gfCNCPoint2[2423] = {X 419.9424, Y 96.5448, Z -2.1667, A 0.000, B 0.000, C 0.000 }
gfCNCPoint2[2424] = {X 419.9467, Y 97.0649, Z -2.1667, A 0.000, B 0.000, C 0.000 }
gfCNCPoint2[2425] = {X 419.9467, Y 98.0000, Z -2.1667, A 0.000, B 0.000, C 0.000 }
gfCNCPoint2[2426] = {X 419.8404, Y 98.9435, Z -2.1667, A 0.000, B 0.000, C 0.000 }
gfCNCPoint2[2427] = {X 419.5268, Y 99.8397, Z -2.1667, A 0.000, B 0.000, C 0.000 }
gfCNCPoint2[2428] = {X 419.0217, Y 100.6436, Z -2.1667, A 0.000, B 0.000, C 0.000 }
gfCNCPoint2[2429] = {X 418.3503, Y 101.3150, Z -2.1667, A 0.000, B 0.000, C 0.000 }
gfCNCPoint2[2430] = {X 417.5464, Y 101.8201, Z -2.1667, A 0.000, B 0.000, C 0.000 }
gfCNCPoint2[2431] = {X 416.6502, Y 102.1337, Z -2.1667, A 0.000, B 0.000, C 0.000 }
gfCNCPoint2[2432] = {X 415.7067, Y 102.2400, Z -2.1667, A 0.000, B 0.000, C 0.000 }
gfCNCPoint2[2433] = {X 396.4059, Y 102.2400, Z -2.1667, A 0.000, B 0.000, C 0.000 }
gfCNCPoint2[2434] = {X 395.4625, Y 102.1337, Z -2.1667, A 0.000, B 0.000, C 0.000 }
gfCNCPoint2[2435] = {X 394.5663, Y 101.8201, Z -2.1667, A 0.000, B 0.000, C 0.000 }
gfCNCPoint2[2436] = {X 393.7624, Y 101.3150, Z -2.1667, A 0.000, B 0.000, C 0.000 }
gfCNCPoint2[2437] = {X 393.0910, Y 100.6436, Z -2.1667, A 0.000, B 0.000, C 0.000 }
gfCNCPoint2[2438] = {X 392.5858, Y 99.8397, Z -2.1667, A 0.000, B 0.000, C 0.000 }
gfCNCPoint2[2439] = {X 392.2723, Y 98.9435, Z -2.1667, A 0.000, B 0.000, C 0.000 }
gfCNCPoint2[2440] = {X 392.1659, Y 98.0000, Z -2.1667, A 0.000, B 0.000, C 0.000 }
gfCNCPoint2[2441] = {X 392.1659, Y 97.0659, Z -2.1667, A 0.000, B 0.000, C 0.000 }
gfCNCPoint2[2442] = {X 392.2718, Y 96.1245, Z -2.1667, A 0.000, B 0.000, C 0.000 }
gfCNCPoint2[2443] = {X 392.5840, Y 95.2301, Z -2.1667, A 0.000, B 0.000, C 0.000 }
gfCNCPoint2[2444] = {X 393.0870, Y 94.4274, Z -2.1667, A 0.000, B 0.000, C 0.000 }
gfCNCPoint2[2445] = {X 393.7556, Y 93.7563, Z -2.1667, A 0.000, B 0.000, C 0.000 }
gfCNCPoint2[2446] = {X 394.5566, Y 93.2505, Z -2.1667, A 0.000, B 0.000, C 0.000 }
gfCNCPoint2[2447] = {X 395.4499, Y 92.9351, Z -2.1667, A 0.000, B 0.000, C 0.000 }
gfCNCPoint2[2448] = {X 396.3909, Y 92.8260, Z -2.1667, A 0.000, B 0.000, C 0.000 }
gfCNCPoint2[2449] = {X 397.3487, Y 92.7854, Z -2.1667, A 0.000, B 0.000, C 0.000 }
gfCNCPoint2[2450] = {X 398.3031, Y 92.6947, Z -2.1667, A 0.000, B 0.000, C 0.000 }
gfCNCPoint2[2451] = {X 398.9716, Y 92.5328, Z -2.1667, A 0.000, B 0.000, C 0.000 }
gfCNCPoint2[2452] = {X 399.5871, Y 92.2258, Z -2.1667, A 0.000, B 0.000, C 0.000 }
gfCNCPoint2[2453] = {X 413.8427, Y 83.0964, Z -2.1667, A 0.000, B 0.000, C 0.000 }
gfCNCPoint2[2454] = {X 411.6855, Y 79.7280, Z -2.1667, A 0.000, B 0.000, C 0.000 }
gfCNCPoint2[2455] = {X 413.8858, Y 83.1638, Z -2.1667, A 0.000, B 0.000, C 0.000 }
gfCNCPoint2[2456] = {X 428.4059, Y 73.8650, Z -2.1667, A 0.000, B 0.000, C 0.000 }
gfCNCPoint2[2457] = {X 403.8140, Y 64.2159, Z -2.1667, A 0.000, B 0.000, C 0.000 }
gfCNCPoint2[2458] = {X 402.1005, Y 63.6486, Z -2.1667, A 0.000, B 0.000, C 0.000 }
gfCNCPoint2[2459] = {X 400.3349, Y 63.2731, Z -2.1667, A 0.000, B 0.000, C 0.000 }
gfCNCPoint2[2460] = {X 398.5388, Y 63.0940, Z -2.1667, A 0.000, B 0.000, C 0.000 }
gfCNCPoint2[2461] = {X 397.6210, Y 62.9872, Z -2.1667, A 0.000, B 0.000, C 0.000 }
gfCNCPoint2[2462] = {X 396.7495, Y 62.6805, Z -2.1667, A 0.000, B 0.000, C 0.000 }
gfCNCPoint2[2463] = {X 395.9671, Y 62.1889, Z -2.1667, A 0.000, B 0.000, C 0.000 }
gfCNCPoint2[2464] = {X 395.3125, Y 61.5368, Z -2.1667, A 0.000, B 0.000, C 0.000 }
gfCNCPoint2[2465] = {X 394.8180, Y 60.7563, Z -2.1667, A 0.000, B 0.000, C 0.000 }
gfCNCPoint2[2466] = {X 394.5081, Y 59.8858, Z -2.1667, A 0.000, B 0.000, C 0.000 }
gfCNCPoint2[2467] = {X 394.3979, Y 58.9684, Z -2.1667, A 0.000, B 0.000, C 0.000 }
gfCNCPoint2[2468] = {X 394.3977, Y 58.0000, Z -2.1667, A 0.000, B 0.000, C 0.000 }
gfCNCPoint2[2469] = {X 394.5020, Y 57.0743, Z -2.1667, A 0.000, B 0.000, C 0.000 }
gfCNCPoint2[2470] = {X 394.8097, Y 56.1950, Z -2.1667, A 0.000, B 0.000, C 0.000 }
gfCNCPoint2[2471] = {X 395.3053, Y 55.4063, Z -2.1667, A 0.000, B 0.000, C 0.000 }
gfCNCPoint2[2472] = {X 395.9640, Y 54.7476, Z -2.1667, A 0.000, B 0.000, C 0.000 }
gfCNCPoint2[2473] = {X 396.7528, Y 54.2520, Z -2.1667, A 0.000, B 0.000, C 0.000 }
gfCNCPoint2[2474] = {X 397.6320, Y 53.9443, Z -2.1667, A 0.000, B 0.000, C 0.000 }
gfCNCPoint2[2475] = {X 398.5577, Y 53.8400, Z -2.1667, A 0.000, B 0.000, C 0.000 }
gfCNCPoint2[2476] = {X 419.4886, Y 53.8400, Z -2.1667, A 0.000, B 0.000, C 0.000 }
gfCNCPoint2[2477] = {X 420.4143, Y 53.9443, Z -2.1667, A 0.000, B 0.000, C 0.000 }
gfCNCPoint2[2478] = {X 421.2936, Y 54.2520, Z -2.1667, A 0.000, B 0.000, C 0.000 }
gfCNCPoint2[2479] = {X 422.0823, Y 54.7476, Z -2.1667, A 0.000, B 0.000, C 0.000 }
gfCNCPoint2[2480] = {X 422.7410, Y 55.4063, Z -2.1667, A 0.000, B 0.000, C 0.000 }
gfCNCPoint2[2481] = {X 423.2366, Y 56.1950, Z -2.1667, A 0.000, B 0.000, C 0.000 }
gfCNCPoint2[2482] = {X 423.5443, Y 57.0743, Z -2.1667, A 0.000, B 0.000, C 0.000 }
gfCNCPoint2[2483] = {X 423.6486, Y 58.0000, Z -2.1667, A 0.000, B 0.000, C 0.000 }
gfCNCPoint2[2484] = {X 423.6486, Y 58.3421, Z -2.1667, A 0.000, B 0.000, C 0.000 }
gfCNCPoint2[2485] = {X 429.5531, Y 60.6433, Z -2.1667, A 0.000, B 0.000, C 0.000 }
gfCNCPoint2[2486] = {X 458.0211, Y 71.9378, Z -2.1667, A 0.000, B 0.000, C 0.000 }
gfCNCPoint2[2487] = {X 458.0212, Y 63.0709, Z -2.1667, A 0.000, B 0.000, C 0.000 }
gfCNCPoint2[2488] = {X 457.9189, Y 63.0588, Z -2.1667, A 0.000, B 0.000, C 0.000 }
gfCNCPoint2[2489] = {X 457.8169, Y 63.0441, Z -2.1667, A 0.000, B 0.000, C 0.000 }
gfCNCPoint2[2490] = {X 456.8792, Y 62.7822, Z -2.1667, A 0.000, B 0.000, C 0.000 }
gfCNCPoint2[2491] = {X 456.0281, Y 62.3095, Z -2.1667, A 0.000, B 0.000, C 0.000 }
gfCNCPoint2[2492] = {X 455.3102, Y 61.6519, Z -2.1667, A 0.000, B 0.000, C 0.000 }
gfCNCPoint2[2493] = {X 454.7647, Y 60.8455, Z -2.1667, A 0.000, B 0.000, C 0.000 }
gfCNCPoint2[2494] = {X 454.4217, Y 59.9343, Z -2.1667, A 0.000, B 0.000, C 0.000 }
gfCNCPoint2[2495] = {X 454.2997, Y 58.9684, Z -2.1667, A 0.000, B 0.000, C 0.000 }
gfCNCPoint2[2496] = {X 454.2996, Y 58.0000, Z -2.1667, A 0.000, B 0.000, C 0.000 }
gfCNCPoint2[2497] = {X 454.4039, Y 57.0743, Z -2.1667, A 0.000, B 0.000, C 0.000 }
gfCNCPoint2[2498] = {X 454.7116, Y 56.1950, Z -2.1667, A 0.000, B 0.000, C 0.000 }
gfCNCPoint2[2499] = {X 455.2072, Y 55.4063, Z -2.1667, A 0.000, B 0.000, C 0.000 }
gfCNCPoint2[2500] = {X 455.8659, Y 54.7476, Z -2.1667, A 0.000, B 0.000, C 0.000 }
gfCNCPoint2[2501] = {X 456.6546, Y 54.2520, Z -2.1667, A 0.000, B 0.000, C 0.000 }
gfCNCPoint2[2502] = {X 457.5339, Y 53.9443, Z -2.1667, A 0.000, B 0.000, C 0.000 }
gfCNCPoint2[2503] = {X 458.4596, Y 53.8400, Z -2.1667, A 0.000, B 0.000, C 0.000 }
gfCNCPoint2[2504] = {X 475.0000, Y 53.8400, Z -2.1667, A 0.000, B 0.000, C 0.000 }
gfCNCPoint2[2505] = {X 475.9257, Y 53.9443, Z -2.1667, A 0.000, B 0.000, C 0.000 }
gfCNCPoint2[2506] = {X 476.8050, Y 54.2520, Z -2.1667, A 0.000, B 0.000, C 0.000 }
gfCNCPoint2[2507] = {X 477.5937, Y 54.7476, Z -2.1667, A 0.000, B 0.000, C 0.000 }
gfCNCPoint2[2508] = {X 478.2524, Y 55.4063, Z -2.1667, A 0.000, B 0.000, C 0.000 }
gfCNCPoint2[2509] = {X 478.7480, Y 56.1950, Z -2.1667, A 0.000, B 0.000, C 0.000 }
gfCNCPoint2[2510] = {X 479.0557, Y 57.0743, Z -2.1667, A 0.000, B 0.000, C 0.000 }
gfCNCPoint2[2511] = {X 479.1600, Y 58.0000, Z -2.1667, A 0.000, B 0.000, C 0.000 }
gfCNCPoint2[2512] = {X 479.1600, Y 58.9342, Z -2.1667, A 0.000, B 0.000, C 0.000 }
gfCNCPoint2[2513] = {X 479.0692, Y 59.7985, Z -2.1667, A 0.000, B 0.000, C 0.000 }
gfCNCPoint2[2514] = {X 478.8008, Y 60.6250, Z -2.1667, A 0.000, B 0.000, C 0.000 }
gfCNCPoint2[2515] = {X 478.3666, Y 61.3777, Z -2.1667, A 0.000, B 0.000, C 0.000 }
gfCNCPoint2[2516] = {X 477.7855, Y 62.0238, Z -2.1667, A 0.000, B 0.000, C 0.000 }
gfCNCPoint2[2517] = {X 477.0828, Y 62.5351, Z -2.1667, A 0.000, B 0.000, C 0.000 }
gfCNCPoint2[2518] = {X 476.2893, Y 62.8892, Z -2.1667, A 0.000, B 0.000, C 0.000 }
gfCNCPoint2[2519] = {X 475.4395, Y 63.0708, Z -2.1667, A 0.000, B 0.000, C 0.000 }
gfCNCPoint2[2520] = {X 475.4399, Y 92.8982, Z -2.1667, A 0.000, B 0.000, C 0.000 }
gfCNCPoint2[2521] = {X 475.8913, Y 93.0052, Z -2.1667, A 0.000, B 0.000, C 0.000 }
gfCNCPoint2[2522] = {X 476.3356, Y 93.1389, Z -2.1667, A 0.000, B 0.000, C 0.000 }
gfCNCPoint2[2523] = {X 477.1173, Y 93.4941, Z -2.1667, A 0.000, B 0.000, C 0.000 }
gfCNCPoint2[2524] = {X 477.8089, Y 94.0030, Z -2.1667, A 0.000, B 0.000, C 0.000 }
gfCNCPoint2[2525] = {X 478.3804, Y 94.6438, Z -2.1667, A 0.000, B 0.000, C 0.000 }
gfCNCPoint2[2526] = {X 478.8072, Y 95.3889, Z -2.1667, A 0.000, B 0.000, C 0.000 }
gfCNCPoint2[2527] = {X 479.0708, Y 96.2060, Z -2.1667, A 0.000, B 0.000, C 0.000 }
gfCNCPoint2[2528] = {X 479.1600, Y 97.0600, Z -2.1667, A 0.000, B 0.000, C 0.000 }
gfCNCPoint2[2529] = {X 479.1600, Y 98.0000, Z -2.1667, A 0.000, B 0.000, C 0.000 }
gfCNCPoint2[2530] = {X 479.0557, Y 98.9257, Z -2.1667, A 0.000, B 0.000, C 0.000 }
gfCNCPoint2[2531] = {X 478.7480, Y 99.8050, Z -2.1667, A 0.000, B 0.000, C 0.000 }
gfCNCPoint2[2532] = {X 478.2524, Y 100.5937, Z -2.1667, A 0.000, B 0.000, C 0.000 }
gfCNCPoint2[2533] = {X 477.5937, Y 101.2524, Z -2.1667, A 0.000, B 0.000, C 0.000 }
gfCNCPoint2[2534] = {X 476.8050, Y 101.7480, Z -2.1667, A 0.000, B 0.000, C 0.000 }
gfCNCPoint2[2535] = {X 475.9257, Y 102.0557, Z -2.1667, A 0.000, B 0.000, C 0.000 }
gfCNCPoint2[2536] = {X 475.0000, Y 102.1600, Z -2.1667, A 0.000, B 0.000, C 0.000 }
gfCNCPoint2[2537] = {X 458.4596, Y 102.1600, Z -2.1667, A 0.000, B 0.000, C 0.000 }
gfCNCPoint2[2538] = {X 457.5339, Y 102.0557, Z -2.1667, A 0.000, B 0.000, C 0.000 }
gfCNCPoint2[2539] = {X 456.6546, Y 101.7480, Z -2.1667, A 0.000, B 0.000, C 0.000 }
gfCNCPoint2[2540] = {X 455.8659, Y 101.2524, Z -2.1667, A 0.000, B 0.000, C 0.000 }
gfCNCPoint2[2541] = {X 455.2072, Y 100.5937, Z -2.1667, A 0.000, B 0.000, C 0.000 }
gfCNCPoint2[2542] = {X 454.7116, Y 99.8050, Z -2.1667, A 0.000, B 0.000, C 0.000 }
gfCNCPoint2[2543] = {X 454.4039, Y 98.9257, Z -2.1667, A 0.000, B 0.000, C 0.000 }
gfCNCPoint2[2544] = {X 454.2996, Y 98.0000, Z -2.1667, A 0.000, B 0.000, C 0.000 }
gfCNCPoint2[2545] = {X 454.2996, Y 97.0659, Z -2.1667, A 0.000, B 0.000, C 0.000 }
gfCNCPoint2[2546] = {X 454.3903, Y 96.2022, Z -2.1667, A 0.000, B 0.000, C 0.000 }
gfCNCPoint2[2547] = {X 454.6583, Y 95.3761, Z -2.1667, A 0.000, B 0.000, C 0.000 }
gfCNCPoint2[2548] = {X 455.0920, Y 94.6237, Z -2.1667, A 0.000, B 0.000, C 0.000 }
gfCNCPoint2[2549] = {X 455.6724, Y 93.9777, Z -2.1667, A 0.000, B 0.000, C 0.000 }
gfCNCPoint2[2550] = {X 456.3743, Y 93.4663, Z -2.1667, A 0.000, B 0.000, C 0.000 }
gfCNCPoint2[2551] = {X 457.1672, Y 93.1118, Z -2.1667, A 0.000, B 0.000, C 0.000 }
gfCNCPoint2[2552] = {X 458.0163, Y 92.9296, Z -2.1667, A 0.000, B 0.000, C 0.000 }
gfCNCPoint2[2553] = {X 458.0163, Y 85.4858, Z -2.1667, A 0.000, B 0.000, C 0.000 }
gfCNCPoint2[2554] = {X 444.8401, Y 80.3207, Z -2.1667, A 0.000, B 0.000, C 0.000 }
gfCNCPoint2[2555] = {X 419.8620, Y 96.5015, Z -2.1667, A 0.000, B 0.000, C 0.000 }
gfCNCPoint2[2556] = {X 419.8667, Y 97.0652, Z -2.1667, A 0.000, B 0.000, C 0.000 }
gfCNCPoint2[2557] = {X 419.8667, Y 98.0000, Z -2.1667, A 0.000, B 0.000, C 0.000 }
gfCNCPoint2[2558] = {X 419.7624, Y 98.9257, Z -2.1667, A 0.000, B 0.000, C 0.000 }
gfCNCPoint2[2559] = {X 419.4547, Y 99.8050, Z -2.1667, A 0.000, B 0.000, C 0.000 }
gfCNCPoint2[2560] = {X 418.9591, Y 100.5937, Z -2.1667, A 0.000, B 0.000, C 0.000 }
gfCNCPoint2[2561] = {X 418.3004, Y 101.2524, Z -2.1667, A 0.000, B 0.000, C 0.000 }
gfCNCPoint2[2562] = {X 417.5117, Y 101.7480, Z -2.1667, A 0.000, B 0.000, C 0.000 }
gfCNCPoint2[2563] = {X 416.6324, Y 102.0557, Z -2.1667, A 0.000, B 0.000, C 0.000 }
gfCNCPoint2[2564] = {X 415.7067, Y 102.1600, Z -2.1667, A 0.000, B 0.000, C 0.000 }
gfCNCPoint2[2565] = {X 396.4059, Y 102.1600, Z -2.1667, A 0.000, B 0.000, C 0.000 }
gfCNCPoint2[2566] = {X 395.4803, Y 102.0557, Z -2.1667, A 0.000, B 0.000, C 0.000 }
gfCNCPoint2[2567] = {X 394.6010, Y 101.7480, Z -2.1667, A 0.000, B 0.000, C 0.000 }
gfCNCPoint2[2568] = {X 393.8122, Y 101.2524, Z -2.1667, A 0.000, B 0.000, C 0.000 }
gfCNCPoint2[2569] = {X 393.1535, Y 100.5937, Z -2.1667, A 0.000, B 0.000, C 0.000 }
gfCNCPoint2[2570] = {X 392.6579, Y 99.8050, Z -2.1667, A 0.000, B 0.000, C 0.000 }
gfCNCPoint2[2571] = {X 392.3502, Y 98.9257, Z -2.1667, A 0.000, B 0.000, C 0.000 }
gfCNCPoint2[2572] = {X 392.2459, Y 98.0000, Z -2.1667, A 0.000, B 0.000, C 0.000 }
gfCNCPoint2[2573] = {X 392.2459, Y 97.0659, Z -2.1667, A 0.000, B 0.000, C 0.000 }
gfCNCPoint2[2574] = {X 392.3498, Y 96.1422, Z -2.1667, A 0.000, B 0.000, C 0.000 }
gfCNCPoint2[2575] = {X 392.6562, Y 95.2646, Z -2.1667, A 0.000, B 0.000, C 0.000 }
gfCNCPoint2[2576] = {X 393.1497, Y 94.4770, Z -2.1667, A 0.000, B 0.000, C 0.000 }
gfCNCPoint2[2577] = {X 393.8059, Y 93.8186, Z -2.1667, A 0.000, B 0.000, C 0.000 }
gfCNCPoint2[2578] = {X 394.5918, Y 93.3223, Z -2.1667, A 0.000, B 0.000, C 0.000 }
gfCNCPoint2[2579] = {X 395.4684, Y 93.0130, Z -2.1667, A 0.000, B 0.000, C 0.000 }
gfCNCPoint2[2580] = {X 396.3917, Y 92.9060, Z -2.1667, A 0.000, B 0.000, C 0.000 }
gfCNCPoint2[2581] = {X 397.3541, Y 92.8652, Z -2.1667, A 0.000, B 0.000, C 0.000 }
gfCNCPoint2[2582] = {X 398.3130, Y 92.7741, Z -2.1667, A 0.000, B 0.000, C 0.000 }
gfCNCPoint2[2583] = {X 398.9990, Y 92.6080, Z -2.1667, A 0.000, B 0.000, C 0.000 }
gfCNCPoint2[2584] = {X 399.6306, Y 92.2929, Z -2.1667, A 0.000, B 0.000, C 0.000 }
gfCNCPoint2[2585] = {X 413.8858, Y 83.1638, Z -2.1667, A 0.000, B 0.000, C 0.000 }
gfCNCPoint2[2586] = {X 411.7287, Y 79.7953, Z -2.1667, A 0.000, B 0.000, C 0.000 }
gfCNCPoint2[2587] = {X 413.9290, Y 83.2312, Z -2.1667, A 0.000, B 0.000, C 0.000 }
gfCNCPoint2[2588] = {X 428.5811, Y 73.8478, Z -2.1667, A 0.000, B 0.000, C 0.000 }
gfCNCPoint2[2589] = {X 403.8433, Y 64.1415, Z -2.1667, A 0.000, B 0.000, C 0.000 }
gfCNCPoint2[2590] = {X 402.1209, Y 63.5713, Z -2.1667, A 0.000, B 0.000, C 0.000 }
gfCNCPoint2[2591] = {X 400.3462, Y 63.1939, Z -2.1667, A 0.000, B 0.000, C 0.000 }
gfCNCPoint2[2592] = {X 398.5408, Y 63.0140, Z -2.1667, A 0.000, B 0.000, C 0.000 }
gfCNCPoint2[2593] = {X 397.6404, Y 62.9096, Z -2.1667, A 0.000, B 0.000, C 0.000 }
gfCNCPoint2[2594] = {X 396.7853, Y 62.6089, Z -2.1667, A 0.000, B 0.000, C 0.000 }
gfCNCPoint2[2595] = {X 396.0176, Y 62.1269, Z -2.1667, A 0.000, B 0.000, C 0.000 }
gfCNCPoint2[2596] = {X 395.3753, Y 61.4873, Z -2.1667, A 0.000, B 0.000, C 0.000 }
gfCNCPoint2[2597] = {X 394.8902, Y 60.7216, Z -2.1667, A 0.000, B 0.000, C 0.000 }
gfCNCPoint2[2598] = {X 394.5860, Y 59.8677, Z -2.1667, A 0.000, B 0.000, C 0.000 }
gfCNCPoint2[2599] = {X 394.4779, Y 58.9678, Z -2.1667, A 0.000, B 0.000, C 0.000 }
gfCNCPoint2[2600] = {X 394.4777, Y 58.0000, Z -2.1667, A 0.000, B 0.000, C 0.000 }
gfCNCPoint2[2601] = {X 394.5800, Y 57.0921, Z -2.1667, A 0.000, B 0.000, C 0.000 }
gfCNCPoint2[2602] = {X 394.8818, Y 56.2298, Z -2.1667, A 0.000, B 0.000, C 0.000 }
gfCNCPoint2[2603] = {X 395.3678, Y 55.4562, Z -2.1667, A 0.000, B 0.000, C 0.000 }
gfCNCPoint2[2604] = {X 396.0139, Y 54.8101, Z -2.1667, A 0.000, B 0.000, C 0.000 }
gfCNCPoint2[2605] = {X 396.7875, Y 54.3240, Z -2.1667, A 0.000, B 0.000, C 0.000 }
gfCNCPoint2[2606] = {X 397.6498, Y 54.0223, Z -2.1667, A 0.000, B 0.000, C 0.000 }
gfCNCPoint2[2607] = {X 398.5577, Y 53.9200, Z -2.1667, A 0.000, B 0.000, C 0.000 }
gfCNCPoint2[2608] = {X 419.4886, Y 53.9200, Z -2.1667, A 0.000, B 0.000, C 0.000 }
gfCNCPoint2[2609] = {X 420.3965, Y 54.0223, Z -2.1667, A 0.000, B 0.000, C 0.000 }
gfCNCPoint2[2610] = {X 421.2589, Y 54.3240, Z -2.1667, A 0.000, B 0.000, C 0.000 }
gfCNCPoint2[2611] = {X 422.0324, Y 54.8101, Z -2.1667, A 0.000, B 0.000, C 0.000 }
gfCNCPoint2[2612] = {X 422.6785, Y 55.4562, Z -2.1667, A 0.000, B 0.000, C 0.000 }
gfCNCPoint2[2613] = {X 423.1646, Y 56.2298, Z -2.1667, A 0.000, B 0.000, C 0.000 }
gfCNCPoint2[2614] = {X 423.4663, Y 57.0921, Z -2.1667, A 0.000, B 0.000, C 0.000 }
gfCNCPoint2[2615] = {X 423.5686, Y 58.0000, Z -2.1667, A 0.000, B 0.000, C 0.000 }
gfCNCPoint2[2616] = {X 423.5686, Y 58.3968, Z -2.1667, A 0.000, B 0.000, C 0.000 }
gfCNCPoint2[2617] = {X 429.5238, Y 60.7177, Z -2.1667, A 0.000, B 0.000, C 0.000 }
gfCNCPoint2[2618] = {X 458.1011, Y 72.0556, Z -2.1667, A 0.000, B 0.000, C 0.000 }
gfCNCPoint2[2619] = {X 458.1012, Y 62.9983, Z -2.1667, A 0.000, B 0.000, C 0.000 }
gfCNCPoint2[2620] = {X 457.9650, Y 62.9840, Z -2.1667, A 0.000, B 0.000, C 0.000 }
gfCNCPoint2[2621] = {X 457.8293, Y 62.9651, Z -2.1667, A 0.000, B 0.000, C 0.000 }
gfCNCPoint2[2622] = {X 456.9096, Y 62.7082, Z -2.1667, A 0.000, B 0.000, C 0.000 }
gfCNCPoint2[2623] = {X 456.0749, Y 62.2446, Z -2.1667, A 0.000, B 0.000, C 0.000 }
gfCNCPoint2[2624] = {X 455.3707, Y 61.5996, Z -2.1667, A 0.000, B 0.000, C 0.000 }
gfCNCPoint2[2625] = {X 454.8358, Y 60.8087, Z -2.1667, A 0.000, B 0.000, C 0.000 }
gfCNCPoint2[2626] = {X 454.4993, Y 59.9151, Z -2.1667, A 0.000, B 0.000, C 0.000 }
gfCNCPoint2[2627] = {X 454.3797, Y 58.9678, Z -2.1667, A 0.000, B 0.000, C 0.000 }
gfCNCPoint2[2628] = {X 454.3796, Y 58.0000, Z -2.1667, A 0.000, B 0.000, C 0.000 }
gfCNCPoint2[2629] = {X 454.4819, Y 57.0921, Z -2.1667, A 0.000, B 0.000, C 0.000 }
gfCNCPoint2[2630] = {X 454.7837, Y 56.2298, Z -2.1667, A 0.000, B 0.000, C 0.000 }
gfCNCPoint2[2631] = {X 455.2697, Y 55.4562, Z -2.1667, A 0.000, B 0.000, C 0.000 }
gfCNCPoint2[2632] = {X 455.9158, Y 54.8101, Z -2.1667, A 0.000, B 0.000, C 0.000 }
gfCNCPoint2[2633] = {X 456.6894, Y 54.3240, Z -2.1667, A 0.000, B 0.000, C 0.000 }
gfCNCPoint2[2634] = {X 457.5517, Y 54.0223, Z -2.1667, A 0.000, B 0.000, C 0.000 }
gfCNCPoint2[2635] = {X 458.4596, Y 53.9200, Z -2.1667, A 0.000, B 0.000, C 0.000 }
gfCNCPoint2[2636] = {X 475.0000, Y 53.9200, Z -2.1667, A 0.000, B 0.000, C 0.000 }
gfCNCPoint2[2637] = {X 475.9079, Y 54.0223, Z -2.1667, A 0.000, B 0.000, C 0.000 }
gfCNCPoint2[2638] = {X 476.7702, Y 54.3240, Z -2.1667, A 0.000, B 0.000, C 0.000 }
gfCNCPoint2[2639] = {X 477.5438, Y 54.8101, Z -2.1667, A 0.000, B 0.000, C 0.000 }
gfCNCPoint2[2640] = {X 478.1899, Y 55.4562, Z -2.1667, A 0.000, B 0.000, C 0.000 }
gfCNCPoint2[2641] = {X 478.6760, Y 56.2298, Z -2.1667, A 0.000, B 0.000, C 0.000 }
gfCNCPoint2[2642] = {X 478.9777, Y 57.0921, Z -2.1667, A 0.000, B 0.000, C 0.000 }
gfCNCPoint2[2643] = {X 479.0800, Y 58.0000, Z -2.1667, A 0.000, B 0.000, C 0.000 }
gfCNCPoint2[2644] = {X 479.0800, Y 58.9342, Z -2.1667, A 0.000, B 0.000, C 0.000 }
gfCNCPoint2[2645] = {X 478.9888, Y 59.7919, Z -2.1667, A 0.000, B 0.000, C 0.000 }
gfCNCPoint2[2646] = {X 478.7194, Y 60.6112, Z -2.1667, A 0.000, B 0.000, C 0.000 }
gfCNCPoint2[2647] = {X 478.2837, Y 61.3556, Z -2.1667, A 0.000, B 0.000, C 0.000 }
gfCNCPoint2[2648] = {X 477.7013, Y 61.9917, Z -2.1667, A 0.000, B 0.000, C 0.000 }
gfCNCPoint2[2649] = {X 476.9982, Y 62.4913, Z -2.1667, A 0.000, B 0.000, C 0.000 }
gfCNCPoint2[2650] = {X 476.2058, Y 62.8318, Z -2.1667, A 0.000, B 0.000, C 0.000 }
gfCNCPoint2[2651] = {X 475.3595, Y 62.9982, Z -2.1667, A 0.000, B 0.000, C 0.000 }
gfCNCPoint2[2652] = {X 475.3599, Y 92.9637, Z -2.1667, A 0.000, B 0.000, C 0.000 }
gfCNCPoint2[2653] = {X 475.8391, Y 93.0740, Z -2.1667, A 0.000, B 0.000, C 0.000 }
gfCNCPoint2[2654] = {X 476.3102, Y 93.2148, Z -2.1667, A 0.000, B 0.000, C 0.000 }
gfCNCPoint2[2655] = {X 477.0769, Y 93.5631, Z -2.1667, A 0.000, B 0.000, C 0.000 }
gfCNCPoint2[2656] = {X 477.7550, Y 94.0622, Z -2.1667, A 0.000, B 0.000, C 0.000 }
gfCNCPoint2[2657] = {X 478.3155, Y 94.6906, Z -2.1667, A 0.000, B 0.000, C 0.000 }
gfCNCPoint2[2658] = {X 478.7340, Y 95.4212, Z -2.1667, A 0.000, B 0.000, C 0.000 }
gfCNCPoint2[2659] = {X 478.9926, Y 96.2226, Z -2.1667, A 0.000, B 0.000, C 0.000 }
gfCNCPoint2[2660] = {X 479.0800, Y 97.0600, Z -2.1667, A 0.000, B 0.000, C 0.000 }
gfCNCPoint2[2661] = {X 479.0800, Y 98.0000, Z -2.1667, A 0.000, B 0.000, C 0.000 }
gfCNCPoint2[2662] = {X 478.9777, Y 98.9079, Z -2.1667, A 0.000, B 0.000, C 0.000 }
gfCNCPoint2[2663] = {X 478.6760, Y 99.7702, Z -2.1667, A 0.000, B 0.000, C 0.000 }
gfCNCPoint2[2664] = {X 478.1899, Y 100.5438, Z -2.1667, A 0.000, B 0.000, C 0.000 }
gfCNCPoint2[2665] = {X 477.5438, Y 101.1899, Z -2.1667, A 0.000, B 0.000, C 0.000 }
gfCNCPoint2[2666] = {X 476.7702, Y 101.6760, Z -2.1667, A 0.000, B 0.000, C 0.000 }
gfCNCPoint2[2667] = {X 475.9079, Y 101.9777, Z -2.1667, A 0.000, B 0.000, C 0.000 }
gfCNCPoint2[2668] = {X 475.0000, Y 102.0800, Z -2.1667, A 0.000, B 0.000, C 0.000 }
gfCNCPoint2[2669] = {X 458.4596, Y 102.0800, Z -2.1667, A 0.000, B 0.000, C 0.000 }
gfCNCPoint2[2670] = {X 457.5517, Y 101.9777, Z -2.1667, A 0.000, B 0.000, C 0.000 }
gfCNCPoint2[2671] = {X 456.6894, Y 101.6760, Z -2.1667, A 0.000, B 0.000, C 0.000 }
gfCNCPoint2[2672] = {X 455.9158, Y 101.1899, Z -2.1667, A 0.000, B 0.000, C 0.000 }
gfCNCPoint2[2673] = {X 455.2697, Y 100.5438, Z -2.1667, A 0.000, B 0.000, C 0.000 }
gfCNCPoint2[2674] = {X 454.7837, Y 99.7702, Z -2.1667, A 0.000, B 0.000, C 0.000 }
gfCNCPoint2[2675] = {X 454.4819, Y 98.9079, Z -2.1667, A 0.000, B 0.000, C 0.000 }
gfCNCPoint2[2676] = {X 454.3796, Y 98.0000, Z -2.1667, A 0.000, B 0.000, C 0.000 }
gfCNCPoint2[2677] = {X 454.3796, Y 97.0659, Z -2.1667, A 0.000, B 0.000, C 0.000 }
gfCNCPoint2[2678] = {X 454.4707, Y 96.2088, Z -2.1667, A 0.000, B 0.000, C 0.000 }
gfCNCPoint2[2679] = {X 454.7398, Y 95.3899, Z -2.1667, A 0.000, B 0.000, C 0.000 }
gfCNCPoint2[2680] = {X 455.1749, Y 94.6458, Z -2.1667, A 0.000, B 0.000, C 0.000 }
gfCNCPoint2[2681] = {X 455.7566, Y 94.0098, Z -2.1667, A 0.000, B 0.000, C 0.000 }
gfCNCPoint2[2682] = {X 456.4590, Y 93.5101, Z -2.1667, A 0.000, B 0.000, C 0.000 }
gfCNCPoint2[2683] = {X 457.2507, Y 93.1692, Z -2.1667, A 0.000, B 0.000, C 0.000 }
gfCNCPoint2[2684] = {X 458.0963, Y 93.0021, Z -2.1667, A 0.000, B 0.000, C 0.000 }
gfCNCPoint2[2685] = {X 458.0963, Y 85.4313, Z -2.1667, A 0.000, B 0.000, C 0.000 }
gfCNCPoint2[2686] = {X 444.8311, Y 80.2313, Z -2.1667, A 0.000, B 0.000, C 0.000 }
gfCNCPoint2[2687] = {X 419.7816, Y 96.4583, Z -2.1667, A 0.000, B 0.000, C 0.000 }
gfCNCPoint2[2688] = {X 419.7867, Y 97.0656, Z -2.1667, A 0.000, B 0.000, C 0.000 }
gfCNCPoint2[2689] = {X 419.7867, Y 98.0000, Z -2.1667, A 0.000, B 0.000, C 0.000 }
gfCNCPoint2[2690] = {X 419.6844, Y 98.9079, Z -2.1667, A 0.000, B 0.000, C 0.000 }
gfCNCPoint2[2691] = {X 419.3827, Y 99.7702, Z -2.1667, A 0.000, B 0.000, C 0.000 }
gfCNCPoint2[2692] = {X 418.8966, Y 100.5438, Z -2.1667, A 0.000, B 0.000, C 0.000 }
gfCNCPoint2[2693] = {X 418.2505, Y 101.1899, Z -2.1667, A 0.000, B 0.000, C 0.000 }
gfCNCPoint2[2694] = {X 417.4769, Y 101.6760, Z -2.1667, A 0.000, B 0.000, C 0.000 }
gfCNCPoint2[2695] = {X 416.6146, Y 101.9777, Z -2.1667, A 0.000, B 0.000, C 0.000 }
gfCNCPoint2[2696] = {X 415.7067, Y 102.0800, Z -2.1667, A 0.000, B 0.000, C 0.000 }
gfCNCPoint2[2697] = {X 396.4059, Y 102.0800, Z -2.1667, A 0.000, B 0.000, C 0.000 }
gfCNCPoint2[2698] = {X 395.4981, Y 101.9777, Z -2.1667, A 0.000, B 0.000, C 0.000 }
gfCNCPoint2[2699] = {X 394.6357, Y 101.6760, Z -2.1667, A 0.000, B 0.000, C 0.000 }
gfCNCPoint2[2700] = {X 393.8621, Y 101.1899, Z -2.1667, A 0.000, B 0.000, C 0.000 }
gfCNCPoint2[2701] = {X 393.2161, Y 100.5438, Z -2.1667, A 0.000, B 0.000, C 0.000 }
gfCNCPoint2[2702] = {X 392.7300, Y 99.7702, Z -2.1667, A 0.000, B 0.000, C 0.000 }
gfCNCPoint2[2703] = {X 392.4282, Y 98.9079, Z -2.1667, A 0.000, B 0.000, C 0.000 }
gfCNCPoint2[2704] = {X 392.3259, Y 98.0000, Z -2.1667, A 0.000, B 0.000, C 0.000 }
gfCNCPoint2[2705] = {X 392.3259, Y 97.0659, Z -2.1667, A 0.000, B 0.000, C 0.000 }
gfCNCPoint2[2706] = {X 392.4278, Y 96.1599, Z -2.1667, A 0.000, B 0.000, C 0.000 }
gfCNCPoint2[2707] = {X 392.7283, Y 95.2991, Z -2.1667, A 0.000, B 0.000, C 0.000 }
gfCNCPoint2[2708] = {X 393.2125, Y 94.5266, Z -2.1667, A 0.000, B 0.000, C 0.000 }
gfCNCPoint2[2709] = {X 393.8561, Y 93.8808, Z -2.1667, A 0.000, B 0.000, C 0.000 }
gfCNCPoint2[2710] = {X 394.6271, Y 93.3942, Z -2.1667, A 0.000, B 0.000, C 0.000 }
gfCNCPoint2[2711] = {X 395.4869, Y 93.0908, Z -2.1667, A 0.000, B 0.000, C 0.000 }
gfCNCPoint2[2712] = {X 396.3925, Y 92.9860, Z -2.1667, A 0.000, B 0.000, C 0.000 }
gfCNCPoint2[2713] = {X 397.3594, Y 92.9450, Z -2.1667, A 0.000, B 0.000, C 0.000 }
gfCNCPoint2[2714] = {X 398.3229, Y 92.8535, Z -2.1667, A 0.000, B 0.000, C 0.000 }
gfCNCPoint2[2715] = {X 399.0264, Y 92.6832, Z -2.1667, A 0.000, B 0.000, C 0.000 }
gfCNCPoint2[2716] = {X 399.6742, Y 92.3601, Z -2.1667, A 0.000, B 0.000, C 0.000 }
gfCNCPoint2[2717] = {X 413.9290, Y 83.2312, Z -2.1667, A 0.000, B 0.000, C 0.000 }
gfCNCPoint2[2718] = {X 411.7653, Y 79.8525, Z -2.1667, A 0.000, B 0.000, C 0.000 }
gfCNCPoint2[2719] = {X 411.7676, Y 79.8510, Z -2.1667, A 0.000, B 0.000, C 0.000 }
gfCNCPoint2[2720] = {X 413.9656, Y 83.2884, Z -2.1667, A 0.000, B 0.000, C 0.000 }
gfCNCPoint2[2721] = {X 428.7564, Y 73.8307, Z -2.1667, A 0.000, B 0.000, C 0.000 }
gfCNCPoint2[2722] = {X 403.8726, Y 64.0670, Z -2.1667, A 0.000, B 0.000, C 0.000 }
gfCNCPoint2[2723] = {X 402.1413, Y 63.4939, Z -2.1667, A 0.000, B 0.000, C 0.000 }
gfCNCPoint2[2724] = {X 400.3575, Y 63.1147, Z -2.1667, A 0.000, B 0.000, C 0.000 }
gfCNCPoint2[2725] = {X 398.5427, Y 62.9340, Z -2.1667, A 0.000, B 0.000, C 0.000 }
gfCNCPoint2[2726] = {X 397.6551, Y 62.8309, Z -2.1667, A 0.000, B 0.000, C 0.000 }
gfCNCPoint2[2727] = {X 396.8125, Y 62.5333, Z -2.1667, A 0.000, B 0.000, C 0.000 }
gfCNCPoint2[2728] = {X 396.0571, Y 62.0560, Z -2.1667, A 0.000, B 0.000, C 0.000 }
gfCNCPoint2[2729] = {X 395.4264, Y 61.4230, Z -2.1667, A 0.000, B 0.000, C 0.000 }
gfCNCPoint2[2730] = {X 394.9520, Y 60.6657, Z -2.1667, A 0.000, B 0.000, C 0.000 }
gfCNCPoint2[2731] = {X 394.6575, Y 59.8220, Z -2.1667, A 0.000, B 0.000, C 0.000 }
gfCNCPoint2[2732] = {X 394.5577, Y 58.9340, Z -2.1667, A 0.000, B 0.000, C 0.000 }
gfCNCPoint2[2733] = {X 394.5577, Y 58.0000, Z -2.1667, A 0.000, B 0.000, C 0.000 }
gfCNCPoint2[2734] = {X 394.6580, Y 57.1099, Z -2.1667, A 0.000, B 0.000, C 0.000 }
gfCNCPoint2[2735] = {X 394.9538, Y 56.2645, Z -2.1667, A 0.000, B 0.000, C 0.000 }
gfCNCPoint2[2736] = {X 395.4304, Y 55.5060, Z -2.1667, A 0.000, B 0.000, C 0.000 }
gfCNCPoint2[2737] = {X 396.0638, Y 54.8727, Z -2.1667, A 0.000, B 0.000, C 0.000 }
gfCNCPoint2[2738] = {X 396.8222, Y 54.3961, Z -2.1667, A 0.000, B 0.000, C 0.000 }
gfCNCPoint2[2739] = {X 397.6676, Y 54.1003, Z -2.1667, A 0.000, B 0.000, C 0.000 }
gfCNCPoint2[2740] = {X 398.5577, Y 54.0000, Z -2.1667, A 0.000, B 0.000, C 0.000 }
gfCNCPoint2[2741] = {X 419.4886, Y 54.0000, Z -2.1667, A 0.000, B 0.000, C 0.000 }
gfCNCPoint2[2742] = {X 420.3787, Y 54.1003, Z -2.1667, A 0.000, B 0.000, C 0.000 }
gfCNCPoint2[2743] = {X 421.2241, Y 54.3961, Z -2.1667, A 0.000, B 0.000, C 0.000 }
gfCNCPoint2[2744] = {X 421.9826, Y 54.8727, Z -2.1667, A 0.000, B 0.000, C 0.000 }
gfCNCPoint2[2745] = {X 422.6159, Y 55.5060, Z -2.1667, A 0.000, B 0.000, C 0.000 }
gfCNCPoint2[2746] = {X 423.0925, Y 56.2645, Z -2.1667, A 0.000, B 0.000, C 0.000 }
gfCNCPoint2[2747] = {X 423.3883, Y 57.1099, Z -2.1667, A 0.000, B 0.000, C 0.000 }
gfCNCPoint2[2748] = {X 423.4886, Y 58.0000, Z -2.1667, A 0.000, B 0.000, C 0.000 }
gfCNCPoint2[2749] = {X 423.4886, Y 58.4514, Z -2.1667, A 0.000, B 0.000, C 0.000 }
gfCNCPoint2[2750] = {X 429.4945, Y 60.7922, Z -2.1667, A 0.000, B 0.000, C 0.000 }
gfCNCPoint2[2751] = {X 458.1791, Y 72.1726, Z -2.1667, A 0.000, B 0.000, C 0.000 }
gfCNCPoint2[2752] = {X 458.1810, Y 71.5843, Z -2.1667, A 0.000, B 0.000, C 0.000 }
gfCNCPoint2[2753] = {X 458.1798, Y 63.0380, Z -2.1667, A 0.000, B 0.000, C 0.000 }
gfCNCPoint2[2754] = {X 458.1841, Y 62.9246, Z -2.1667, A 0.000, B 0.000, C 0.000 }
gfCNCPoint2[2755] = {X 458.0124, Y 62.9090, Z -2.1667, A 0.000, B 0.000, C 0.000 }
gfCNCPoint2[2756] = {X 457.8416, Y 62.8860, Z -2.1667, A 0.000, B 0.000, C 0.000 }
gfCNCPoint2[2757] = {X 456.9349, Y 62.6321, Z -2.1667, A 0.000, B 0.000, C 0.000 }
gfCNCPoint2[2758] = {X 456.1127, Y 62.1732, Z -2.1667, A 0.000, B 0.000, C 0.000 }
gfCNCPoint2[2759] = {X 455.4205, Y 61.5348, Z -2.1667, A 0.000, B 0.000, C 0.000 }
gfCNCPoint2[2760] = {X 454.8968, Y 60.7524, Z -2.1667, A 0.000, B 0.000, C 0.000 }
gfCNCPoint2[2761] = {X 454.5704, Y 59.8691, Z -2.1667, A 0.000, B 0.000, C 0.000 }
gfCNCPoint2[2762] = {X 454.4596, Y 58.9340, Z -2.1667, A 0.000, B 0.000, C 0.000 }
gfCNCPoint2[2763] = {X 454.4596, Y 58.0000, Z -2.1667, A 0.000, B 0.000, C 0.000 }
gfCNCPoint2[2764] = {X 454.5599, Y 57.1099, Z -2.1667, A 0.000, B 0.000, C 0.000 }
gfCNCPoint2[2765] = {X 454.8557, Y 56.2645, Z -2.1667, A 0.000, B 0.000, C 0.000 }
gfCNCPoint2[2766] = {X 455.3323, Y 55.5060, Z -2.1667, A 0.000, B 0.000, C 0.000 }
gfCNCPoint2[2767] = {X 455.9656, Y 54.8727, Z -2.1667, A 0.000, B 0.000, C 0.000 }
gfCNCPoint2[2768] = {X 456.7241, Y 54.3961, Z -2.1667, A 0.000, B 0.000, C 0.000 }
gfCNCPoint2[2769] = {X 457.5695, Y 54.1003, Z -2.1667, A 0.000, B 0.000, C 0.000 }
gfCNCPoint2[2770] = {X 458.4596, Y 54.0000, Z -2.1667, A 0.000, B 0.000, C 0.000 }
gfCNCPoint2[2771] = {X 475.0000, Y 54.0000, Z -2.1667, A 0.000, B 0.000, C 0.000 }
gfCNCPoint2[2772] = {X 475.8901, Y 54.1003, Z -2.1667, A 0.000, B 0.000, C 0.000 }
gfCNCPoint2[2773] = {X 476.7355, Y 54.3961, Z -2.1667, A 0.000, B 0.000, C 0.000 }
gfCNCPoint2[2774] = {X 477.4940, Y 54.8727, Z -2.1667, A 0.000, B 0.000, C 0.000 }
gfCNCPoint2[2775] = {X 478.1273, Y 55.5060, Z -2.1667, A 0.000, B 0.000, C 0.000 }
gfCNCPoint2[2776] = {X 478.6039, Y 56.2645, Z -2.1667, A 0.000, B 0.000, C 0.000 }
gfCNCPoint2[2777] = {X 478.8997, Y 57.1099, Z -2.1667, A 0.000, B 0.000, C 0.000 }
gfCNCPoint2[2778] = {X 479.0000, Y 58.0000, Z -2.1667, A 0.000, B 0.000, C 0.000 }
gfCNCPoint2[2779] = {X 478.9999, Y 58.9671, Z -2.1667, A 0.000, B 0.000, C 0.000 }
gfCNCPoint2[2780] = {X 478.9023, Y 59.8128, Z -2.1667, A 0.000, B 0.000, C 0.000 }
gfCNCPoint2[2781] = {X 478.6280, Y 60.6187, Z -2.1667, A 0.000, B 0.000, C 0.000 }
gfCNCPoint2[2782] = {X 478.1893, Y 61.3483, Z -2.1667, A 0.000, B 0.000, C 0.000 }
gfCNCPoint2[2783] = {X 477.6062, Y 61.9685, Z -2.1667, A 0.000, B 0.000, C 0.000 }
gfCNCPoint2[2784] = {X 476.9050, Y 62.4513, Z -2.1667, A 0.000, B 0.000, C 0.000 }
gfCNCPoint2[2785] = {X 476.1175, Y 62.7748, Z -2.1667, A 0.000, B 0.000, C 0.000 }
gfCNCPoint2[2786] = {X 475.2795, Y 62.9243, Z -2.1667, A 0.000, B 0.000, C 0.000 }
gfCNCPoint2[2787] = {X 475.2799, Y 93.0297, Z -2.1667, A 0.000, B 0.000, C 0.000 }
gfCNCPoint2[2788] = {X 475.7868, Y 93.1431, Z -2.1667, A 0.000, B 0.000, C 0.000 }
gfCNCPoint2[2789] = {X 476.2849, Y 93.2907, Z -2.1667, A 0.000, B 0.000, C 0.000 }
gfCNCPoint2[2790] = {X 477.0364, Y 93.6321, Z -2.1667, A 0.000, B 0.000, C 0.000 }
gfCNCPoint2[2791] = {X 477.7012, Y 94.1213, Z -2.1667, A 0.000, B 0.000, C 0.000 }
gfCNCPoint2[2792] = {X 478.2505, Y 94.7373, Z -2.1667, A 0.000, B 0.000, C 0.000 }
gfCNCPoint2[2793] = {X 478.6608, Y 95.4536, Z -2.1667, A 0.000, B 0.000, C 0.000 }
gfCNCPoint2[2794] = {X 478.9143, Y 96.2391, Z -2.1667, A 0.000, B 0.000, C 0.000 }
gfCNCPoint2[2795] = {X 479.0000, Y 97.0600, Z -2.1667, A 0.000, B 0.000, C 0.000 }
gfCNCPoint2[2796] = {X 479.0000, Y 98.0000, Z -2.1667, A 0.000, B 0.000, C 0.000 }
gfCNCPoint2[2797] = {X 478.8997, Y 98.8901, Z -2.1667, A 0.000, B 0.000, C 0.000 }
gfCNCPoint2[2798] = {X 478.6039, Y 99.7355, Z -2.1667, A 0.000, B 0.000, C 0.000 }
gfCNCPoint2[2799] = {X 478.1273, Y 100.4940, Z -2.1667, A 0.000, B 0.000, C 0.000 }
gfCNCPoint2[2800] = {X 477.4940, Y 101.1273, Z -2.1667, A 0.000, B 0.000, C 0.000 }
gfCNCPoint2[2801] = {X 476.7355, Y 101.6039, Z -2.1667, A 0.000, B 0.000, C 0.000 }
gfCNCPoint2[2802] = {X 475.8901, Y 101.8997, Z -2.1667, A 0.000, B 0.000, C 0.000 }
gfCNCPoint2[2803] = {X 475.0000, Y 102.0000, Z -2.1667, A 0.000, B 0.000, C 0.000 }
gfCNCPoint2[2804] = {X 458.4596, Y 102.0000, Z -2.1667, A 0.000, B 0.000, C 0.000 }
gfCNCPoint2[2805] = {X 457.5695, Y 101.8997, Z -2.1667, A 0.000, B 0.000, C 0.000 }
gfCNCPoint2[2806] = {X 456.7241, Y 101.6039, Z -2.1667, A 0.000, B 0.000, C 0.000 }
gfCNCPoint2[2807] = {X 455.9656, Y 101.1273, Z -2.1667, A 0.000, B 0.000, C 0.000 }
gfCNCPoint2[2808] = {X 455.3323, Y 100.4940, Z -2.1667, A 0.000, B 0.000, C 0.000 }
gfCNCPoint2[2809] = {X 454.8557, Y 99.7355, Z -2.1667, A 0.000, B 0.000, C 0.000 }
gfCNCPoint2[2810] = {X 454.5599, Y 98.8901, Z -2.1667, A 0.000, B 0.000, C 0.000 }
gfCNCPoint2[2811] = {X 454.4596, Y 98.0000, Z -2.1667, A 0.000, B 0.000, C 0.000 }
gfCNCPoint2[2812] = {X 454.4596, Y 97.0659, Z -2.1667, A 0.000, B 0.000, C 0.000 }
gfCNCPoint2[2813] = {X 454.5511, Y 96.2154, Z -2.1667, A 0.000, B 0.000, C 0.000 }
gfCNCPoint2[2814] = {X 454.8213, Y 95.4037, Z -2.1667, A 0.000, B 0.000, C 0.000 }
gfCNCPoint2[2815] = {X 455.2580, Y 94.6681, Z -2.1667, A 0.000, B 0.000, C 0.000 }
gfCNCPoint2[2816] = {X 455.8411, Y 94.0422, Z -2.1667, A 0.000, B 0.000, C 0.000 }
gfCNCPoint2[2817] = {X 456.5439, Y 93.5545, Z -2.1667, A 0.000, B 0.000, C 0.000 }
gfCNCPoint2[2818] = {X 457.3344, Y 93.2275, Z -2.1667, A 0.000, B 0.000, C 0.000 }
gfCNCPoint2[2819] = {X 458.1763, Y 93.0760, Z -2.1667, A 0.000, B 0.000, C 0.000 }
gfCNCPoint2[2820] = {X 458.1763, Y 85.3767, Z -2.1667, A 0.000, B 0.000, C 0.000 }
gfCNCPoint2[2821] = {X 445.0132, Y 80.2167, Z -2.1667, A 0.000, B 0.000, C 0.000 }
gfCNCPoint2[2822] = {X 444.8210, Y 80.1425, Z -2.1667, A 0.000, B 0.000, C 0.000 }
gfCNCPoint2[2823] = {X 419.7013, Y 96.4150, Z -2.1667, A 0.000, B 0.000, C 0.000 }
gfCNCPoint2[2824] = {X 419.7067, Y 97.0659, Z -2.1667, A 0.000, B 0.000, C 0.000 }
gfCNCPoint2[2825] = {X 419.7067, Y 98.0000, Z -2.1667, A 0.000, B 0.000, C 0.000 }
gfCNCPoint2[2826] = {X 419.6064, Y 98.8901, Z -2.1667, A 0.000, B 0.000, C 0.000 }
gfCNCPoint2[2827] = {X 419.3106, Y 99.7355, Z -2.1667, A 0.000, B 0.000, C 0.000 }
gfCNCPoint2[2828] = {X 418.8340, Y 100.4940, Z -2.1667, A 0.000, B 0.000, C 0.000 }
gfCNCPoint2[2829] = {X 418.2007, Y 101.1273, Z -2.1667, A 0.000, B 0.000, C 0.000 }
gfCNCPoint2[2830] = {X 417.4422, Y 101.6039, Z -2.1667, A 0.000, B 0.000, C 0.000 }
gfCNCPoint2[2831] = {X 416.5968, Y 101.8997, Z -2.1667, A 0.000, B 0.000, C 0.000 }
gfCNCPoint2[2832] = {X 415.7067, Y 102.0000, Z -2.1667, A 0.000, B 0.000, C 0.000 }
gfCNCPoint2[2833] = {X 396.4059, Y 102.0000, Z -2.1667, A 0.000, B 0.000, C 0.000 }
gfCNCPoint2[2834] = {X 395.5159, Y 101.8997, Z -2.1667, A 0.000, B 0.000, C 0.000 }
gfCNCPoint2[2835] = {X 394.6704, Y 101.6039, Z -2.1667, A 0.000, B 0.000, C 0.000 }
gfCNCPoint2[2836] = {X 393.9120, Y 101.1273, Z -2.1667, A 0.000, B 0.000, C 0.000 }
gfCNCPoint2[2837] = {X 393.2786, Y 100.4940, Z -2.1667, A 0.000, B 0.000, C 0.000 }
gfCNCPoint2[2838] = {X 392.8021, Y 99.7355, Z -2.1667, A 0.000, B 0.000, C 0.000 }
gfCNCPoint2[2839] = {X 392.5062, Y 98.8901, Z -2.1667, A 0.000, B 0.000, C 0.000 }
gfCNCPoint2[2840] = {X 392.4059, Y 98.0000, Z -2.1667, A 0.000, B 0.000, C 0.000 }
gfCNCPoint2[2841] = {X 392.4059, Y 97.0659, Z -2.1667, A 0.000, B 0.000, C 0.000 }
gfCNCPoint2[2842] = {X 392.5058, Y 96.1776, Z -2.1667, A 0.000, B 0.000, C 0.000 }
gfCNCPoint2[2843] = {X 392.8005, Y 95.3337, Z -2.1667, A 0.000, B 0.000, C 0.000 }
gfCNCPoint2[2844] = {X 393.2753, Y 94.5762, Z -2.1667, A 0.000, B 0.000, C 0.000 }
gfCNCPoint2[2845] = {X 393.9064, Y 93.9431, Z -2.1667, A 0.000, B 0.000, C 0.000 }
gfCNCPoint2[2846] = {X 394.6623, Y 93.4660, Z -2.1667, A 0.000, B 0.000, C 0.000 }
gfCNCPoint2[2847] = {X 395.5053, Y 93.1686, Z -2.1667, A 0.000, B 0.000, C 0.000 }
gfCNCPoint2[2848] = {X 396.3933, Y 93.0660, Z -2.1667, A 0.000, B 0.000, C 0.000 }
gfCNCPoint2[2849] = {X 397.3648, Y 93.0249, Z -2.1667, A 0.000, B 0.000, C 0.000 }
gfCNCPoint2[2850] = {X 398.3327, Y 92.9329, Z -2.1667, A 0.000, B 0.000, C 0.000 }
gfCNCPoint2[2851] = {X 399.0538, Y 92.7583, Z -2.1667, A 0.000, B 0.000, C 0.000 }
gfCNCPoint2[2852] = {X 399.7177, Y 92.4272, Z -2.1667, A 0.000, B 0.000, C 0.000 }
gfCNCPoint2[2853] = {X 405.3932, Y 88.7698, Z -2.1667, A 0.000, B 0.000, C 0.000 }
gfCNCPoint2[2854] = {X 413.9656, Y 83.2884, Z -2.1667, A 0.000, B 0.000, C 0.000 }
gfCNCPoint2[2855] = {X 411.7676, Y 79.8510, Z -2.1667, A 0.000, B 0.000, C 0.000 }
gfCNCPoint2[2856] = {X 411.7676, Y 79.8510, Z 0.8333, A 0.000, B 0.000, C 0.000 }
gfCNCPoint2[2857] = {X 411.7676, Y 79.8510, Z 11.0000, A 0.000, B 0.000, C 0.000 }
gfCNCPoint2[2858] = {X 466.3099, Y 28.5935, Z 11.0000, A 0.000, B 0.000, C 0.000 }
gfCNCPoint2[2859] = {X 466.3099, Y 28.5935, Z 0.8333, A 0.000, B 0.000, C 0.000 }
gfCNCPoint2[2860] = {X 466.3099, Y 28.5935, Z -2.1667, A 0.000, B 0.000, C 0.000 }
gfCNCPoint2[2861] = {X 462.2299, Y 28.5936, Z -2.1667, A 0.000, B 0.000, C 0.000 }
gfCNCPoint2[2862] = {X 462.2301, Y 40.9128, Z -2.1667, A 0.000, B 0.000, C 0.000 }
gfCNCPoint2[2863] = {X 462.2389, Y 40.9199, Z -2.1667, A 0.000, B 0.000, C 0.000 }
gfCNCPoint2[2864] = {X 462.8740, Y 41.5904, Z -2.1667, A 0.000, B 0.000, C 0.000 }
gfCNCPoint2[2865] = {X 463.3520, Y 42.3806, Z -2.1667, A 0.000, B 0.000, C 0.000 }
gfCNCPoint2[2866] = {X 463.6512, Y 43.2544, Z -2.1667, A 0.000, B 0.000, C 0.000 }
gfCNCPoint2[2867] = {X 463.7578, Y 44.1718, Z -2.1667, A 0.000, B 0.000, C 0.000 }
gfCNCPoint2[2868] = {X 463.7579, Y 45.0000, Z -2.1667, A 0.000, B 0.000, C 0.000 }
gfCNCPoint2[2869] = {X 463.6496, Y 45.9613, Z -2.1667, A 0.000, B 0.000, C 0.000 }
gfCNCPoint2[2870] = {X 463.3301, Y 46.8744, Z -2.1667, A 0.000, B 0.000, C 0.000 }
gfCNCPoint2[2871] = {X 462.8155, Y 47.6935, Z -2.1667, A 0.000, B 0.000, C 0.000 }
gfCNCPoint2[2872] = {X 462.1314, Y 48.3775, Z -2.1667, A 0.000, B 0.000, C 0.000 }
gfCNCPoint2[2873] = {X 461.3123, Y 48.8922, Z -2.1667, A 0.000, B 0.000, C 0.000 }
gfCNCPoint2[2874] = {X 460.3992, Y 49.2117, Z -2.1667, A 0.000, B 0.000, C 0.000 }
gfCNCPoint2[2875] = {X 459.4379, Y 49.3200, Z -2.1667, A 0.000, B 0.000, C 0.000 }
gfCNCPoint2[2876] = {X 452.9945, Y 49.3200, Z -2.1667, A 0.000, B 0.000, C 0.000 }
gfCNCPoint2[2877] = {X 452.0380, Y 49.2128, Z -2.1667, A 0.000, B 0.000, C 0.000 }
gfCNCPoint2[2878] = {X 451.1291, Y 48.8965, Z -2.1667, A 0.000, B 0.000, C 0.000 }
gfCNCPoint2[2879] = {X 450.3127, Y 48.3868, Z -2.1667, A 0.000, B 0.000, C 0.000 }
gfCNCPoint2[2880] = {X 449.6294, Y 47.7091, Z -2.1667, A 0.000, B 0.000, C 0.000 }
gfCNCPoint2[2881] = {X 449.1132, Y 46.8968, Z -2.1667, A 0.000, B 0.000, C 0.000 }
gfCNCPoint2[2882] = {X 448.7895, Y 45.9905, Z -2.1667, A 0.000, B 0.000, C 0.000 }
gfCNCPoint2[2883] = {X 448.6746, Y 45.0349, Z -2.1667, A 0.000, B 0.000, C 0.000 }
gfCNCPoint2[2884] = {X 448.6749, Y 44.1494, Z -2.1667, A 0.000, B 0.000, C 0.000 }
gfCNCPoint2[2885] = {X 448.7853, Y 43.2364, Z -2.1667, A 0.000, B 0.000, C 0.000 }
gfCNCPoint2[2886] = {X 449.0865, Y 42.3675, Z -2.1667, A 0.000, B 0.000, C 0.000 }
gfCNCPoint2[2887] = {X 449.5648, Y 41.5821, Z -2.1667, A 0.000, B 0.000, C 0.000 }
gfCNCPoint2[2888] = {X 450.1984, Y 40.9157, Z -2.1667, A 0.000, B 0.000, C 0.000 }
gfCNCPoint2[2889] = {X 450.1984, Y 34.4738, Z -2.1667, A 0.000, B 0.000, C 0.000 }
gfCNCPoint2[2890] = {X 447.4737, Y 34.4738, Z -2.1667, A 0.000, B 0.000, C 0.000 }
gfCNCPoint2[2891] = {X 443.1892, Y 42.8156, Z -2.1667, A 0.000, B 0.000, C 0.000 }
gfCNCPoint2[2892] = {X 443.1943, Y 42.8293, Z -2.1667, A 0.000, B 0.000, C 0.000 }
gfCNCPoint2[2893] = {X 443.3604, Y 43.4909, Z -2.1667, A 0.000, B 0.000, C 0.000 }
gfCNCPoint2[2894] = {X 443.4203, Y 44.1703, Z -2.1667, A 0.000, B 0.000, C 0.000 }
gfCNCPoint2[2895] = {X 443.4205, Y 45.0000, Z -2.1667, A 0.000, B 0.000, C 0.000 }
gfCNCPoint2[2896] = {X 443.3122, Y 45.9613, Z -2.1667, A 0.000, B 0.000, C 0.000 }
gfCNCPoint2[2897] = {X 442.9927, Y 46.8744, Z -2.1667, A 0.000, B 0.000, C 0.000 }
gfCNCPoint2[2898] = {X 442.4780, Y 47.6935, Z -2.1667, A 0.000, B 0.000, C 0.000 }
gfCNCPoint2[2899] = {X 441.7939, Y 48.3775, Z -2.1667, A 0.000, B 0.000, C 0.000 }
gfCNCPoint2[2900] = {X 440.9748, Y 48.8922, Z -2.1667, A 0.000, B 0.000, C 0.000 }
gfCNCPoint2[2901] = {X 440.0618, Y 49.2117, Z -2.1667, A 0.000, B 0.000, C 0.000 }
gfCNCPoint2[2902] = {X 439.1005, Y 49.3200, Z -2.1667, A 0.000, B 0.000, C 0.000 }
gfCNCPoint2[2903] = {X 432.5144, Y 49.3200, Z -2.1667, A 0.000, B 0.000, C 0.000 }
gfCNCPoint2[2904] = {X 431.5531, Y 49.2117, Z -2.1667, A 0.000, B 0.000, C 0.000 }
gfCNCPoint2[2905] = {X 430.6401, Y 48.8922, Z -2.1667, A 0.000, B 0.000, C 0.000 }
gfCNCPoint2[2906] = {X 429.8210, Y 48.3775, Z -2.1667, A 0.000, B 0.000, C 0.000 }
gfCNCPoint2[2907] = {X 429.1369, Y 47.6935, Z -2.1667, A 0.000, B 0.000, C 0.000 }
gfCNCPoint2[2908] = {X 428.6223, Y 46.8745, Z -2.1667, A 0.000, B 0.000, C 0.000 }
gfCNCPoint2[2909] = {X 428.3027, Y 45.9614, Z -2.1667, A 0.000, B 0.000, C 0.000 }
gfCNCPoint2[2910] = {X 428.1944, Y 45.0001, Z -2.1667, A 0.000, B 0.000, C 0.000 }
gfCNCPoint2[2911] = {X 428.1948, Y 44.1494, Z -2.1667, A 0.000, B 0.000, C 0.000 }
gfCNCPoint2[2912] = {X 428.2925, Y 43.2935, Z -2.1667, A 0.000, B 0.000, C 0.000 }
gfCNCPoint2[2913] = {X 428.5580, Y 42.4740, Z -2.1667, A 0.000, B 0.000, C 0.000 }
gfCNCPoint2[2914] = {X 428.9809, Y 41.7236, Z -2.1667, A 0.000, B 0.000, C 0.000 }
gfCNCPoint2[2915] = {X 429.5442, Y 41.0719, Z -2.1667, A 0.000, B 0.000, C 0.000 }
gfCNCPoint2[2916] = {X 430.2256, Y 40.5449, Z -2.1667, A 0.000, B 0.000, C 0.000 }
gfCNCPoint2[2917] = {X 430.9981, Y 40.1637, Z -2.1667, A 0.000, B 0.000, C 0.000 }
gfCNCPoint2[2918] = {X 434.9874, Y 32.3550, Z -2.1667, A 0.000, B 0.000, C 0.000 }
gfCNCPoint2[2919] = {X 433.8176, Y 31.5685, Z -2.1667, A 0.000, B 0.000, C 0.000 }
gfCNCPoint2[2920] = {X 432.7546, Y 30.6427, Z -2.1667, A 0.000, B 0.000, C 0.000 }
gfCNCPoint2[2921] = {X 431.8149, Y 29.5921, Z -2.1667, A 0.000, B 0.000, C 0.000 }
gfCNCPoint2[2922] = {X 431.0130, Y 28.4327, Z -2.1667, A 0.000, B 0.000, C 0.000 }
gfCNCPoint2[2923] = {X 430.3614, Y 27.1828, Z -2.1667, A 0.000, B 0.000, C 0.000 }
gfCNCPoint2[2924] = {X 429.8703, Y 25.8615, Z -2.1667, A 0.000, B 0.000, C 0.000 }
gfCNCPoint2[2925] = {X 429.4511, Y 24.0500, Z -2.1667, A 0.000, B 0.000, C 0.000 }
gfCNCPoint2[2926] = {X 429.2376, Y 22.2029, Z -2.1667, A 0.000, B 0.000, C 0.000 }
gfCNCPoint2[2927] = {X 429.2322, Y 20.3435, Z -2.1667, A 0.000, B 0.000, C 0.000 }
gfCNCPoint2[2928] = {X 429.4351, Y 18.4953, Z -2.1667, A 0.000, B 0.000, C 0.000 }
gfCNCPoint2[2929] = {X 429.8437, Y 16.6814, Z -2.1667, A 0.000, B 0.000, C 0.000 }
gfCNCPoint2[2930] = {X 430.3651, Y 15.2116, Z -2.1667, A 0.000, B 0.000, C 0.000 }
gfCNCPoint2[2931] = {X 431.0759, Y 13.8235, Z -2.1667, A 0.000, B 0.000, C 0.000 }
gfCNCPoint2[2932] = {X 431.9637, Y 12.5414, Z -2.1667, A 0.000, B 0.000, C 0.000 }
gfCNCPoint2[2933] = {X 433.0129, Y 11.3876, Z -2.1667, A 0.000, B 0.000, C 0.000 }
gfCNCPoint2[2934] = {X 434.2051, Y 10.3823, Z -2.1667, A 0.000, B 0.000, C 0.000 }
gfCNCPoint2[2935] = {X 435.5196, Y 9.5431, Z -2.1667, A 0.000, B 0.000, C 0.000 }
gfCNCPoint2[2936] = {X 436.9333, Y 8.8848, Z -2.1667, A 0.000, B 0.000, C 0.000 }
gfCNCPoint2[2937] = {X 438.4216, Y 8.4187, Z -2.1667, A 0.000, B 0.000, C 0.000 }
gfCNCPoint2[2938] = {X 440.0467, Y 8.1097, Z -2.1667, A 0.000, B 0.000, C 0.000 }
gfCNCPoint2[2939] = {X 441.6910, Y 7.9283, Z -2.1667, A 0.000, B 0.000, C 0.000 }
gfCNCPoint2[2940] = {X 443.3444, Y 7.8756, Z -2.1667, A 0.000, B 0.000, C 0.000 }
gfCNCPoint2[2941] = {X 444.0357, Y 7.8716, Z -2.1667, A 0.000, B 0.000, C 0.000 }
gfCNCPoint2[2942] = {X 459.4465, Y 7.8716, Z -2.1667, A 0.000, B 0.000, C 0.000 }
gfCNCPoint2[2943] = {X 460.4059, Y 7.9797, Z -2.1667, A 0.000, B 0.000, C 0.000 }
gfCNCPoint2[2944] = {X 461.3172, Y 8.2985, Z -2.1667, A 0.000, B 0.000, C 0.000 }
gfCNCPoint2[2945] = {X 462.1347, Y 8.8122, Z -2.1667, A 0.000, B 0.000, C 0.000 }
gfCNCPoint2[2946] = {X 462.8173, Y 9.4949, Z -2.1667, A 0.000, B 0.000, C 0.000 }
gfCNCPoint2[2947] = {X 463.3310, Y 10.3123, Z -2.1667, A 0.000, B 0.000, C 0.000 }
gfCNCPoint2[2948] = {X 463.6498, Y 11.2236, Z -2.1667, A 0.000, B 0.000, C 0.000 }
gfCNCPoint2[2949] = {X 463.7579, Y 12.1830, Z -2.1667, A 0.000, B 0.000, C 0.000 }
gfCNCPoint2[2950] = {X 463.7579, Y 12.9781, Z -2.1667, A 0.000, B 0.000, C 0.000 }
gfCNCPoint2[2951] = {X 463.6565, Y 13.9082, Z -2.1667, A 0.000, B 0.000, C 0.000 }
gfCNCPoint2[2952] = {X 463.3572, Y 14.7947, Z -2.1667, A 0.000, B 0.000, C 0.000 }
gfCNCPoint2[2953] = {X 462.8741, Y 15.5959, Z -2.1667, A 0.000, B 0.000, C 0.000 }
gfCNCPoint2[2954] = {X 462.2297, Y 16.2743, Z -2.1667, A 0.000, B 0.000, C 0.000 }
gfCNCPoint2[2955] = {X 462.2299, Y 28.5936, Z -2.1667, A 0.000, B 0.000, C 0.000 }
gfCNCPoint2[2956] = {X 466.2299, Y 28.5935, Z -2.1667, A 0.000, B 0.000, C 0.000 }
gfCNCPoint2[2957] = {X 462.1499, Y 28.5936, Z -2.1667, A 0.000, B 0.000, C 0.000 }
gfCNCPoint2[2958] = {X 462.1501, Y 40.9510, Z -2.1667, A 0.000, B 0.000, C 0.000 }
gfCNCPoint2[2959] = {X 462.1879, Y 40.9815, Z -2.1667, A 0.000, B 0.000, C 0.000 }
gfCNCPoint2[2960] = {X 462.8108, Y 41.6395, Z -2.1667, A 0.000, B 0.000, C 0.000 }
gfCNCPoint2[2961] = {X 463.2798, Y 42.4150, Z -2.1667, A 0.000, B 0.000, C 0.000 }
gfCNCPoint2[2962] = {X 463.5732, Y 43.2723, Z -2.1667, A 0.000, B 0.000, C 0.000 }
gfCNCPoint2[2963] = {X 463.6778, Y 44.1724, Z -2.1667, A 0.000, B 0.000, C 0.000 }
gfCNCPoint2[2964] = {X 463.6779, Y 45.0000, Z -2.1667, A 0.000, B 0.000, C 0.000 }
gfCNCPoint2[2965] = {X 463.5716, Y 45.9435, Z -2.1667, A 0.000, B 0.000, C 0.000 }
gfCNCPoint2[2966] = {X 463.2580, Y 46.8397, Z -2.1667, A 0.000, B 0.000, C 0.000 }
gfCNCPoint2[2967] = {X 462.7529, Y 47.6436, Z -2.1667, A 0.000, B 0.000, C 0.000 }
gfCNCPoint2[2968] = {X 462.0815, Y 48.3150, Z -2.1667, A 0.000, B 0.000, C 0.000 }
gfCNCPoint2[2969] = {X 461.2776, Y 48.8201, Z -2.1667, A 0.000, B 0.000, C 0.000 }
gfCNCPoint2[2970] = {X 460.3814, Y 49.1337, Z -2.1667, A 0.000, B 0.000, C 0.000 }
gfCNCPoint2[2971] = {X 459.4379, Y 49.2400, Z -2.1667, A 0.000, B 0.000, C 0.000 }
gfCNCPoint2[2972] = {X 452.9945, Y 49.2400, Z -2.1667, A 0.000, B 0.000, C 0.000 }
gfCNCPoint2[2973] = {X 452.0558, Y 49.1348, Z -2.1667, A 0.000, B 0.000, C 0.000 }
gfCNCPoint2[2974] = {X 451.1636, Y 48.8243, Z -2.1667, A 0.000, B 0.000, C 0.000 }
gfCNCPoint2[2975] = {X 450.3624, Y 48.3241, Z -2.1667, A 0.000, B 0.000, C 0.000 }
gfCNCPoint2[2976] = {X 449.6918, Y 47.6589, Z -2.1667, A 0.000, B 0.000, C 0.000 }
gfCNCPoint2[2977] = {X 449.1851, Y 46.8617, Z -2.1667, A 0.000, B 0.000, C 0.000 }
gfCNCPoint2[2978] = {X 448.8674, Y 45.9721, Z -2.1667, A 0.000, B 0.000, C 0.000 }
gfCNCPoint2[2979] = {X 448.7546, Y 45.0343, Z -2.1667, A 0.000, B 0.000, C 0.000 }
gfCNCPoint2[2980] = {X 448.7549, Y 44.1505, Z -2.1667, A 0.000, B 0.000, C 0.000 }
gfCNCPoint2[2981] = {X 448.8654, Y 43.2454, Z -2.1667, A 0.000, B 0.000, C 0.000 }
gfCNCPoint2[2982] = {X 449.1668, Y 42.3850, Z -2.1667, A 0.000, B 0.000, C 0.000 }
gfCNCPoint2[2983] = {X 449.6452, Y 41.6088, Z -2.1667, A 0.000, B 0.000, C 0.000 }
gfCNCPoint2[2984] = {X 450.2784, Y 40.9529, Z -2.1667, A 0.000, B 0.000, C 0.000 }
gfCNCPoint2[2985] = {X 450.2784, Y 34.3938, Z -2.1667, A 0.000, B 0.000, C 0.000 }
gfCNCPoint2[2986] = {X 447.4248, Y 34.3938, Z -2.1667, A 0.000, B 0.000, C 0.000 }
gfCNCPoint2[2987] = {X 443.1019, Y 42.8105, Z -2.1667, A 0.000, B 0.000, C 0.000 }
gfCNCPoint2[2988] = {X 443.1189, Y 42.8561, Z -2.1667, A 0.000, B 0.000, C 0.000 }
gfCNCPoint2[2989] = {X 443.2816, Y 43.5048, Z -2.1667, A 0.000, B 0.000, C 0.000 }
gfCNCPoint2[2990] = {X 443.3403, Y 44.1710, Z -2.1667, A 0.000, B 0.000, C 0.000 }
gfCNCPoint2[2991] = {X 443.3405, Y 45.0000, Z -2.1667, A 0.000, B 0.000, C 0.000 }
gfCNCPoint2[2992] = {X 443.2342, Y 45.9435, Z -2.1667, A 0.000, B 0.000, C 0.000 }
gfCNCPoint2[2993] = {X 442.9206, Y 46.8397, Z -2.1667, A 0.000, B 0.000, C 0.000 }
gfCNCPoint2[2994] = {X 442.4154, Y 47.6436, Z -2.1667, A 0.000, B 0.000, C 0.000 }
gfCNCPoint2[2995] = {X 441.7441, Y 48.3150, Z -2.1667, A 0.000, B 0.000, C 0.000 }
gfCNCPoint2[2996] = {X 440.9401, Y 48.8201, Z -2.1667, A 0.000, B 0.000, C 0.000 }
gfCNCPoint2[2997] = {X 440.0440, Y 49.1337, Z -2.1667, A 0.000, B 0.000, C 0.000 }
gfCNCPoint2[2998] = {X 439.1005, Y 49.2400, Z -2.1667, A 0.000, B 0.000, C 0.000 }
gfCNCPoint2[2999] = {X 432.5144, Y 49.2400, Z -2.1667, A 0.000, B 0.000, C 0.000 }
gfCNCPoint2[3000] = {X 431.5709, Y 49.1337, Z -2.1667, A 0.000, B 0.000, C 0.000 }
gfCNCPoint2[3001] = {X 430.6748, Y 48.8201, Z -2.1667, A 0.000, B 0.000, C 0.000 }
gfCNCPoint2[3002] = {X 429.8708, Y 48.3150, Z -2.1667, A 0.000, B 0.000, C 0.000 }
gfCNCPoint2[3003] = {X 429.1995, Y 47.6436, Z -2.1667, A 0.000, B 0.000, C 0.000 }
gfCNCPoint2[3004] = {X 428.6943, Y 46.8397, Z -2.1667, A 0.000, B 0.000, C 0.000 }
gfCNCPoint2[3005] = {X 428.3807, Y 45.9436, Z -2.1667, A 0.000, B 0.000, C 0.000 }
gfCNCPoint2[3006] = {X 428.2744, Y 45.0001, Z -2.1667, A 0.000, B 0.000, C 0.000 }
gfCNCPoint2[3007] = {X 428.2748, Y 44.1505, Z -2.1667, A 0.000, B 0.000, C 0.000 }
gfCNCPoint2[3008] = {X 428.3718, Y 43.3054, Z -2.1667, A 0.000, B 0.000, C 0.000 }
gfCNCPoint2[3009] = {X 428.6354, Y 42.4967, Z -2.1667, A 0.000, B 0.000, C 0.000 }
gfCNCPoint2[3010] = {X 429.0552, Y 41.7570, Z -2.1667, A 0.000, B 0.000, C 0.000 }
gfCNCPoint2[3011] = {X 429.6142, Y 41.1158, Z -2.1667, A 0.000, B 0.000, C 0.000 }
gfCNCPoint2[3012] = {X 430.2899, Y 40.5992, Z -2.1667, A 0.000, B 0.000, C 0.000 }
gfCNCPoint2[3013] = {X 431.0551, Y 40.2278, Z -2.1667, A 0.000, B 0.000, C 0.000 }
gfCNCPoint2[3014] = {X 435.0931, Y 32.3239, Z -2.1667, A 0.000, B 0.000, C 0.000 }
gfCNCPoint2[3015] = {X 433.9163, Y 31.5432, Z -2.1667, A 0.000, B 0.000, C 0.000 }
gfCNCPoint2[3016] = {X 432.8467, Y 30.6211, Z -2.1667, A 0.000, B 0.000, C 0.000 }
gfCNCPoint2[3017] = {X 431.9011, Y 29.5722, Z -2.1667, A 0.000, B 0.000, C 0.000 }
gfCNCPoint2[3018] = {X 431.0945, Y 28.4130, Z -2.1667, A 0.000, B 0.000, C 0.000 }
gfCNCPoint2[3019] = {X 430.4397, Y 27.1618, Z -2.1667, A 0.000, B 0.000, C 0.000 }
gfCNCPoint2[3020] = {X 429.9468, Y 25.8383, Z -2.1667, A 0.000, B 0.000, C 0.000 }
gfCNCPoint2[3021] = {X 429.5299, Y 24.0357, Z -2.1667, A 0.000, B 0.000, C 0.000 }
gfCNCPoint2[3022] = {X 429.3174, Y 22.1977, Z -2.1667, A 0.000, B 0.000, C 0.000 }
gfCNCPoint2[3023] = {X 429.3121, Y 20.3474, Z -2.1667, A 0.000, B 0.000, C 0.000 }
gfCNCPoint2[3024] = {X 429.5140, Y 18.5082, Z -2.1667, A 0.000, B 0.000, C 0.000 }
gfCNCPoint2[3025] = {X 429.9207, Y 16.7032, Z -2.1667, A 0.000, B 0.000, C 0.000 }
gfCNCPoint2[3026] = {X 430.4385, Y 15.2434, Z -2.1667, A 0.000, B 0.000, C 0.000 }
gfCNCPoint2[3027] = {X 431.1445, Y 13.8647, Z -2.1667, A 0.000, B 0.000, C 0.000 }
gfCNCPoint2[3028] = {X 432.0262, Y 12.5912, Z -2.1667, A 0.000, B 0.000, C 0.000 }
gfCNCPoint2[3029] = {X 433.0683, Y 11.4452, Z -2.1667, A 0.000, B 0.000, C 0.000 }
gfCNCPoint2[3030] = {X 434.2525, Y 10.4467, Z -2.1667, A 0.000, B 0.000, C 0.000 }
gfCNCPoint2[3031] = {X 435.5581, Y 9.6133, Z -2.1667, A 0.000, B 0.000, C 0.000 }
gfCNCPoint2[3032] = {X 436.9622, Y 8.9594, Z -2.1667, A 0.000, B 0.000, C 0.000 }
gfCNCPoint2[3033] = {X 438.4404, Y 8.4965, Z -2.1667, A 0.000, B 0.000, C 0.000 }
gfCNCPoint2[3034] = {X 440.0593, Y 8.1887, Z -2.1667, A 0.000, B 0.000, C 0.000 }
gfCNCPoint2[3035] = {X 441.6972, Y 8.0080, Z -2.1667, A 0.000, B 0.000, C 0.000 }
gfCNCPoint2[3036] = {X 443.3443, Y 7.9556, Z -2.1667, A 0.000, B 0.000, C 0.000 }
gfCNCPoint2[3037] = {X 444.0360, Y 7.9516, Z -2.1667, A 0.000, B 0.000, C 0.000 }
gfCNCPoint2[3038] = {X 459.4465, Y 7.9516, Z -2.1667, A 0.000, B 0.000, C 0.000 }
gfCNCPoint2[3039] = {X 460.3881, Y 8.0577, Z -2.1667, A 0.000, B 0.000, C 0.000 }
gfCNCPoint2[3040] = {X 461.2825, Y 8.3706, Z -2.1667, A 0.000, B 0.000, C 0.000 }
gfCNCPoint2[3041] = {X 462.0848, Y 8.8747, Z -2.1667, A 0.000, B 0.000, C 0.000 }
gfCNCPoint2[3042] = {X 462.7548, Y 9.5447, Z -2.1667, A 0.000, B 0.000, C 0.000 }
gfCNCPoint2[3043] = {X 463.2589, Y 10.3470, Z -2.1667, A 0.000, B 0.000, C 0.000 }
gfCNCPoint2[3044] = {X 463.5719, Y 11.2414, Z -2.1667, A 0.000, B 0.000, C 0.000 }
gfCNCPoint2[3045] = {X 463.6779, Y 12.1830, Z -2.1667, A 0.000, B 0.000, C 0.000 }
gfCNCPoint2[3046] = {X 463.6779, Y 12.9781, Z -2.1667, A 0.000, B 0.000, C 0.000 }
gfCNCPoint2[3047] = {X 463.5764, Y 13.9000, Z -2.1667, A 0.000, B 0.000, C 0.000 }
gfCNCPoint2[3048] = {X 463.2768, Y 14.7778, Z -2.1667, A 0.000, B 0.000, C 0.000 }
gfCNCPoint2[3049] = {X 462.7936, Y 15.5694, Z -2.1667, A 0.000, B 0.000, C 0.000 }
gfCNCPoint2[3050] = {X 462.1497, Y 16.2370, Z -2.1667, A 0.000, B 0.000, C 0.000 }
gfCNCPoint2[3051] = {X 462.1499, Y 28.5936, Z -2.1667, A 0.000, B 0.000, C 0.000 }
gfCNCPoint2[3052] = {X 466.1499, Y 28.5935, Z -2.1667, A 0.000, B 0.000, C 0.000 }
gfCNCPoint2[3053] = {X 462.0699, Y 28.5936, Z -2.1667, A 0.000, B 0.000, C 0.000 }
gfCNCPoint2[3054] = {X 462.0701, Y 40.9893, Z -2.1667, A 0.000, B 0.000, C 0.000 }
gfCNCPoint2[3055] = {X 462.1368, Y 41.0431, Z -2.1667, A 0.000, B 0.000, C 0.000 }
gfCNCPoint2[3056] = {X 462.7477, Y 41.6886, Z -2.1667, A 0.000, B 0.000, C 0.000 }
gfCNCPoint2[3057] = {X 463.2075, Y 42.4493, Z -2.1667, A 0.000, B 0.000, C 0.000 }
gfCNCPoint2[3058] = {X 463.4953, Y 43.2902, Z -2.1667, A 0.000, B 0.000, C 0.000 }
gfCNCPoint2[3059] = {X 463.5978, Y 44.1731, Z -2.1667, A 0.000, B 0.000, C 0.000 }
gfCNCPoint2[3060] = {X 463.5979, Y 45.0000, Z -2.1667, A 0.000, B 0.000, C 0.000 }
gfCNCPoint2[3061] = {X 463.4936, Y 45.9257, Z -2.1667, A 0.000, B 0.000, C 0.000 }
gfCNCPoint2[3062] = {X 463.1860, Y 46.8050, Z -2.1667, A 0.000, B 0.000, C 0.000 }
gfCNCPoint2[3063] = {X 462.6904, Y 47.5937, Z -2.1667, A 0.000, B 0.000, C 0.000 }
gfCNCPoint2[3064] = {X 462.0317, Y 48.2524, Z -2.1667, A 0.000, B 0.000, C 0.000 }
gfCNCPoint2[3065] = {X 461.2429, Y 48.7480, Z -2.1667, A 0.000, B 0.000, C 0.000 }
gfCNCPoint2[3066] = {X 460.3636, Y 49.0557, Z -2.1667, A 0.000, B 0.000, C 0.000 }
gfCNCPoint2[3067] = {X 459.4379, Y 49.1600, Z -2.1667, A 0.000, B 0.000, C 0.000 }
gfCNCPoint2[3068] = {X 452.9945, Y 49.1600, Z -2.1667, A 0.000, B 0.000, C 0.000 }
gfCNCPoint2[3069] = {X 452.0735, Y 49.0568, Z -2.1667, A 0.000, B 0.000, C 0.000 }
gfCNCPoint2[3070] = {X 451.1982, Y 48.7522, Z -2.1667, A 0.000, B 0.000, C 0.000 }
gfCNCPoint2[3071] = {X 450.4120, Y 48.2614, Z -2.1667, A 0.000, B 0.000, C 0.000 }
gfCNCPoint2[3072] = {X 449.7541, Y 47.6087, Z -2.1667, A 0.000, B 0.000, C 0.000 }
gfCNCPoint2[3073] = {X 449.2569, Y 46.8266, Z -2.1667, A 0.000, B 0.000, C 0.000 }
gfCNCPoint2[3074] = {X 448.9453, Y 45.9538, Z -2.1667, A 0.000, B 0.000, C 0.000 }
gfCNCPoint2[3075] = {X 448.8346, Y 45.0336, Z -2.1667, A 0.000, B 0.000, C 0.000 }
gfCNCPoint2[3076] = {X 448.8349, Y 44.1516, Z -2.1667, A 0.000, B 0.000, C 0.000 }
gfCNCPoint2[3077] = {X 448.9454, Y 43.2545, Z -2.1667, A 0.000, B 0.000, C 0.000 }
gfCNCPoint2[3078] = {X 449.2471, Y 42.4026, Z -2.1667, A 0.000, B 0.000, C 0.000 }
gfCNCPoint2[3079] = {X 449.7256, Y 41.6358, Z -2.1667, A 0.000, B 0.000, C 0.000 }
gfCNCPoint2[3080] = {X 450.3584, Y 40.9906, Z -2.1667, A 0.000, B 0.000, C 0.000 }
gfCNCPoint2[3081] = {X 450.3584, Y 34.3138, Z -2.1667, A 0.000, B 0.000, C 0.000 }
gfCNCPoint2[3082] = {X 447.3760, Y 34.3138, Z -2.1667, A 0.000, B 0.000, C 0.000 }
gfCNCPoint2[3083] = {X 443.0146, Y 42.8053, Z -2.1667, A 0.000, B 0.000, C 0.000 }
gfCNCPoint2[3084] = {X 443.0435, Y 42.8828, Z -2.1667, A 0.000, B 0.000, C 0.000 }
gfCNCPoint2[3085] = {X 443.2028, Y 43.5187, Z -2.1667, A 0.000, B 0.000, C 0.000 }
gfCNCPoint2[3086] = {X 443.2603, Y 44.1717, Z -2.1667, A 0.000, B 0.000, C 0.000 }
gfCNCPoint2[3087] = {X 443.2605, Y 45.0000, Z -2.1667, A 0.000, B 0.000, C 0.000 }
gfCNCPoint2[3088] = {X 443.1562, Y 45.9257, Z -2.1667, A 0.000, B 0.000, C 0.000 }
gfCNCPoint2[3089] = {X 442.8485, Y 46.8050, Z -2.1667, A 0.000, B 0.000, C 0.000 }
gfCNCPoint2[3090] = {X 442.3529, Y 47.5937, Z -2.1667, A 0.000, B 0.000, C 0.000 }
gfCNCPoint2[3091] = {X 441.6942, Y 48.2524, Z -2.1667, A 0.000, B 0.000, C 0.000 }
gfCNCPoint2[3092] = {X 440.9054, Y 48.7480, Z -2.1667, A 0.000, B 0.000, C 0.000 }
gfCNCPoint2[3093] = {X 440.0262, Y 49.0557, Z -2.1667, A 0.000, B 0.000, C 0.000 }
gfCNCPoint2[3094] = {X 439.1005, Y 49.1600, Z -2.1667, A 0.000, B 0.000, C 0.000 }
gfCNCPoint2[3095] = {X 432.5144, Y 49.1600, Z -2.1667, A 0.000, B 0.000, C 0.000 }
gfCNCPoint2[3096] = {X 431.5887, Y 49.0557, Z -2.1667, A 0.000, B 0.000, C 0.000 }
gfCNCPoint2[3097] = {X 430.7095, Y 48.7480, Z -2.1667, A 0.000, B 0.000, C 0.000 }
gfCNCPoint2[3098] = {X 429.9207, Y 48.2524, Z -2.1667, A 0.000, B 0.000, C 0.000 }
gfCNCPoint2[3099] = {X 429.2620, Y 47.5937, Z -2.1667, A 0.000, B 0.000, C 0.000 }
gfCNCPoint2[3100] = {X 428.7664, Y 46.8050, Z -2.1667, A 0.000, B 0.000, C 0.000 }
gfCNCPoint2[3101] = {X 428.4587, Y 45.9257, Z -2.1667, A 0.000, B 0.000, C 0.000 }
gfCNCPoint2[3102] = {X 428.3544, Y 45.0000, Z -2.1667, A 0.000, B 0.000, C 0.000 }
gfCNCPoint2[3103] = {X 428.3548, Y 44.1516, Z -2.1667, A 0.000, B 0.000, C 0.000 }
gfCNCPoint2[3104] = {X 428.4510, Y 43.3174, Z -2.1667, A 0.000, B 0.000, C 0.000 }
gfCNCPoint2[3105] = {X 428.7128, Y 42.5195, Z -2.1667, A 0.000, B 0.000, C 0.000 }
gfCNCPoint2[3106] = {X 429.1295, Y 41.7905, Z -2.1667, A 0.000, B 0.000, C 0.000 }
gfCNCPoint2[3107] = {X 429.6841, Y 41.1600, Z -2.1667, A 0.000, B 0.000, C 0.000 }
gfCNCPoint2[3108] = {X 430.3541, Y 40.6537, Z -2.1667, A 0.000, B 0.000, C 0.000 }
gfCNCPoint2[3109] = {X 431.1120, Y 40.2923, Z -2.1667, A 0.000, B 0.000, C 0.000 }
gfCNCPoint2[3110] = {X 435.1991, Y 32.2923, Z -2.1667, A 0.000, B 0.000, C 0.000 }
gfCNCPoint2[3111] = {X 434.0152, Y 31.5176, Z -2.1667, A 0.000, B 0.000, C 0.000 }
gfCNCPoint2[3112] = {X 432.9389, Y 30.5993, Z -2.1667, A 0.000, B 0.000, C 0.000 }
gfCNCPoint2[3113] = {X 431.9875, Y 29.5522, Z -2.1667, A 0.000, B 0.000, C 0.000 }
gfCNCPoint2[3114] = {X 431.1761, Y 28.3931, Z -2.1667, A 0.000, B 0.000, C 0.000 }
gfCNCPoint2[3115] = {X 430.5179, Y 27.1408, Z -2.1667, A 0.000, B 0.000, C 0.000 }
gfCNCPoint2[3116] = {X 430.0234, Y 25.8152, Z -2.1667, A 0.000, B 0.000, C 0.000 }
gfCNCPoint2[3117] = {X 429.6086, Y 24.0214, Z -2.1667, A 0.000, B 0.000, C 0.000 }
gfCNCPoint2[3118] = {X 429.3972, Y 22.1924, Z -2.1667, A 0.000, B 0.000, C 0.000 }
gfCNCPoint2[3119] = {X 429.3920, Y 20.3513, Z -2.1667, A 0.000, B 0.000, C 0.000 }
gfCNCPoint2[3120] = {X 429.5930, Y 18.5212, Z -2.1667, A 0.000, B 0.000, C 0.000 }
gfCNCPoint2[3121] = {X 429.9976, Y 16.7251, Z -2.1667, A 0.000, B 0.000, C 0.000 }
gfCNCPoint2[3122] = {X 430.5119, Y 15.2752, Z -2.1667, A 0.000, B 0.000, C 0.000 }
gfCNCPoint2[3123] = {X 431.2131, Y 13.9059, Z -2.1667, A 0.000, B 0.000, C 0.000 }
gfCNCPoint2[3124] = {X 432.0888, Y 12.6411, Z -2.1667, A 0.000, B 0.000, C 0.000 }
gfCNCPoint2[3125] = {X 433.1238, Y 11.5029, Z -2.1667, A 0.000, B 0.000, C 0.000 }
gfCNCPoint2[3126] = {X 434.2999, Y 10.5112, Z -2.1667, A 0.000, B 0.000, C 0.000 }
gfCNCPoint2[3127] = {X 435.5965, Y 9.6834, Z -2.1667, A 0.000, B 0.000, C 0.000 }
gfCNCPoint2[3128] = {X 436.9911, Y 9.0340, Z -2.1667, A 0.000, B 0.000, C 0.000 }
gfCNCPoint2[3129] = {X 438.4592, Y 8.5742, Z -2.1667, A 0.000, B 0.000, C 0.000 }
gfCNCPoint2[3130] = {X 440.0719, Y 8.2677, Z -2.1667, A 0.000, B 0.000, C 0.000 }
gfCNCPoint2[3131] = {X 441.7035, Y 8.0878, Z -2.1667, A 0.000, B 0.000, C 0.000 }
gfCNCPoint2[3132] = {X 443.3443, Y 8.0356, Z -2.1667, A 0.000, B 0.000, C 0.000 }
gfCNCPoint2[3133] = {X 444.0362, Y 8.0316, Z -2.1667, A 0.000, B 0.000, C 0.000 }
gfCNCPoint2[3134] = {X 459.4465, Y 8.0316, Z -2.1667, A 0.000, B 0.000, C 0.000 }
gfCNCPoint2[3135] = {X 460.3703, Y 8.1357, Z -2.1667, A 0.000, B 0.000, C 0.000 }
gfCNCPoint2[3136] = {X 461.2478, Y 8.4427, Z -2.1667, A 0.000, B 0.000, C 0.000 }
gfCNCPoint2[3137] = {X 462.0349, Y 8.9373, Z -2.1667, A 0.000, B 0.000, C 0.000 }
gfCNCPoint2[3138] = {X 462.6922, Y 9.5946, Z -2.1667, A 0.000, B 0.000, C 0.000 }
gfCNCPoint2[3139] = {X 463.1868, Y 10.3817, Z -2.1667, A 0.000, B 0.000, C 0.000 }
gfCNCPoint2[3140] = {X 463.4939, Y 11.2592, Z -2.1667, A 0.000, B 0.000, C 0.000 }
gfCNCPoint2[3141] = {X 463.5979, Y 12.1830, Z -2.1667, A 0.000, B 0.000, C 0.000 }
gfCNCPoint2[3142] = {X 463.5979, Y 12.9781, Z -2.1667, A 0.000, B 0.000, C 0.000 }
gfCNCPoint2[3143] = {X 463.5022, Y 13.8653, Z -2.1667, A 0.000, B 0.000, C 0.000 }
gfCNCPoint2[3144] = {X 463.2195, Y 14.7117, Z -2.1667, A 0.000, B 0.000, C 0.000 }
gfCNCPoint2[3145] = {X 462.7627, Y 15.4784, Z -2.1667, A 0.000, B 0.000, C 0.000 }
gfCNCPoint2[3146] = {X 462.1529, Y 16.1299, Z -2.1667, A 0.000, B 0.000, C 0.000 }
gfCNCPoint2[3147] = {X 462.0697, Y 16.1997, Z -2.1667, A 0.000, B 0.000, C 0.000 }
gfCNCPoint2[3148] = {X 462.0699, Y 28.5936, Z -2.1667, A 0.000, B 0.000, C 0.000 }
gfCNCPoint2[3149] = {X 466.0699, Y 28.5935, Z -2.1667, A 0.000, B 0.000, C 0.000 }
gfCNCPoint2[3150] = {X 461.9899, Y 28.5936, Z -2.1667, A 0.000, B 0.000, C 0.000 }
gfCNCPoint2[3151] = {X 461.9901, Y 41.0275, Z -2.1667, A 0.000, B 0.000, C 0.000 }
gfCNCPoint2[3152] = {X 462.0857, Y 41.1046, Z -2.1667, A 0.000, B 0.000, C 0.000 }
gfCNCPoint2[3153] = {X 462.6845, Y 41.7377, Z -2.1667, A 0.000, B 0.000, C 0.000 }
gfCNCPoint2[3154] = {X 463.1353, Y 42.4836, Z -2.1667, A 0.000, B 0.000, C 0.000 }
gfCNCPoint2[3155] = {X 463.4173, Y 43.3082, Z -2.1667, A 0.000, B 0.000, C 0.000 }
gfCNCPoint2[3156] = {X 463.5178, Y 44.1738, Z -2.1667, A 0.000, B 0.000, C 0.000 }
gfCNCPoint2[3157] = {X 463.5179, Y 45.0000, Z -2.1667, A 0.000, B 0.000, C 0.000 }
gfCNCPoint2[3158] = {X 463.4156, Y 45.9079, Z -2.1667, A 0.000, B 0.000, C 0.000 }
gfCNCPoint2[3159] = {X 463.1139, Y 46.7702, Z -2.1667, A 0.000, B 0.000, C 0.000 }
gfCNCPoint2[3160] = {X 462.6278, Y 47.5438, Z -2.1667, A 0.000, B 0.000, C 0.000 }
gfCNCPoint2[3161] = {X 461.9818, Y 48.1899, Z -2.1667, A 0.000, B 0.000, C 0.000 }
gfCNCPoint2[3162] = {X 461.2082, Y 48.6760, Z -2.1667, A 0.000, B 0.000, C 0.000 }
gfCNCPoint2[3163] = {X 460.3458, Y 48.9777, Z -2.1667, A 0.000, B 0.000, C 0.000 }
gfCNCPoint2[3164] = {X 459.4379, Y 49.0800, Z -2.1667, A 0.000, B 0.000, C 0.000 }
gfCNCPoint2[3165] = {X 452.9945, Y 49.0800, Z -2.1667, A 0.000, B 0.000, C 0.000 }
gfCNCPoint2[3166] = {X 452.0912, Y 48.9788, Z -2.1667, A 0.000, B 0.000, C 0.000 }
gfCNCPoint2[3167] = {X 451.2327, Y 48.6800, Z -2.1667, A 0.000, B 0.000, C 0.000 }
gfCNCPoint2[3168] = {X 450.4617, Y 48.1987, Z -2.1667, A 0.000, B 0.000, C 0.000 }
gfCNCPoint2[3169] = {X 449.8164, Y 47.5585, Z -2.1667, A 0.000, B 0.000, C 0.000 }
gfCNCPoint2[3170] = {X 449.3288, Y 46.7914, Z -2.1667, A 0.000, B 0.000, C 0.000 }
gfCNCPoint2[3171] = {X 449.0232, Y 45.9354, Z -2.1667, A 0.000, B 0.000, C 0.000 }
gfCNCPoint2[3172] = {X 448.9146, Y 45.0330, Z -2.1667, A 0.000, B 0.000, C 0.000 }
gfCNCPoint2[3173] = {X 448.9149, Y 44.1527, Z -2.1667, A 0.000, B 0.000, C 0.000 }
gfCNCPoint2[3174] = {X 449.0254, Y 43.2637, Z -2.1667, A 0.000, B 0.000, C 0.000 }
gfCNCPoint2[3175] = {X 449.3274, Y 42.4203, Z -2.1667, A 0.000, B 0.000, C 0.000 }
gfCNCPoint2[3176] = {X 449.8061, Y 41.6631, Z -2.1667, A 0.000, B 0.000, C 0.000 }
gfCNCPoint2[3177] = {X 450.4384, Y 41.0287, Z -2.1667, A 0.000, B 0.000, C 0.000 }
gfCNCPoint2[3178] = {X 450.4384, Y 34.2338, Z -2.1667, A 0.000, B 0.000, C 0.000 }
gfCNCPoint2[3179] = {X 447.3271, Y 34.2338, Z -2.1667, A 0.000, B 0.000, C 0.000 }
gfCNCPoint2[3180] = {X 442.9273, Y 42.8002, Z -2.1667, A 0.000, B 0.000, C 0.000 }
gfCNCPoint2[3181] = {X 442.9681, Y 42.9095, Z -2.1667, A 0.000, B 0.000, C 0.000 }
gfCNCPoint2[3182] = {X 443.1240, Y 43.5326, Z -2.1667, A 0.000, B 0.000, C 0.000 }
gfCNCPoint2[3183] = {X 443.1803, Y 44.1725, Z -2.1667, A 0.000, B 0.000, C 0.000 }
gfCNCPoint2[3184] = {X 443.1805, Y 45.0000, Z -2.1667, A 0.000, B 0.000, C 0.000 }
gfCNCPoint2[3185] = {X 443.0782, Y 45.9079, Z -2.1667, A 0.000, B 0.000, C 0.000 }
gfCNCPoint2[3186] = {X 442.7764, Y 46.7702, Z -2.1667, A 0.000, B 0.000, C 0.000 }
gfCNCPoint2[3187] = {X 442.2903, Y 47.5438, Z -2.1667, A 0.000, B 0.000, C 0.000 }
gfCNCPoint2[3188] = {X 441.6443, Y 48.1899, Z -2.1667, A 0.000, B 0.000, C 0.000 }
gfCNCPoint2[3189] = {X 440.8707, Y 48.6760, Z -2.1667, A 0.000, B 0.000, C 0.000 }
gfCNCPoint2[3190] = {X 440.0084, Y 48.9777, Z -2.1667, A 0.000, B 0.000, C 0.000 }
gfCNCPoint2[3191] = {X 439.1005, Y 49.0800, Z -2.1667, A 0.000, B 0.000, C 0.000 }
gfCNCPoint2[3192] = {X 432.5144, Y 49.0800, Z -2.1667, A 0.000, B 0.000, C 0.000 }
gfCNCPoint2[3193] = {X 431.6065, Y 48.9777, Z -2.1667, A 0.000, B 0.000, C 0.000 }
gfCNCPoint2[3194] = {X 430.7442, Y 48.6760, Z -2.1667, A 0.000, B 0.000, C 0.000 }
gfCNCPoint2[3195] = {X 429.9706, Y 48.1899, Z -2.1667, A 0.000, B 0.000, C 0.000 }
gfCNCPoint2[3196] = {X 429.3245, Y 47.5438, Z -2.1667, A 0.000, B 0.000, C 0.000 }
gfCNCPoint2[3197] = {X 428.8385, Y 46.7702, Z -2.1667, A 0.000, B 0.000, C 0.000 }
gfCNCPoint2[3198] = {X 428.5367, Y 45.9079, Z -2.1667, A 0.000, B 0.000, C 0.000 }
gfCNCPoint2[3199] = {X 428.4344, Y 45.0000, Z -2.1667, A 0.000, B 0.000, C 0.000 }
gfCNCPoint2[3200] = {X 428.4348, Y 44.1527, Z -2.1667, A 0.000, B 0.000, C 0.000 }
gfCNCPoint2[3201] = {X 428.5303, Y 43.3294, Z -2.1667, A 0.000, B 0.000, C 0.000 }
gfCNCPoint2[3202] = {X 428.7902, Y 42.5424, Z -2.1667, A 0.000, B 0.000, C 0.000 }
gfCNCPoint2[3203] = {X 429.2038, Y 41.8242, Z -2.1667, A 0.000, B 0.000, C 0.000 }
gfCNCPoint2[3204] = {X 429.7540, Y 41.2044, Z -2.1667, A 0.000, B 0.000, C 0.000 }
gfCNCPoint2[3205] = {X 430.4181, Y 40.7085, Z -2.1667, A 0.000, B 0.000, C 0.000 }
gfCNCPoint2[3206] = {X 431.1687, Y 40.3571, Z -2.1667, A 0.000, B 0.000, C 0.000 }
gfCNCPoint2[3207] = {X 435.3053, Y 32.2603, Z -2.1667, A 0.000, B 0.000, C 0.000 }
gfCNCPoint2[3208] = {X 434.1144, Y 31.4916, Z -2.1667, A 0.000, B 0.000, C 0.000 }
gfCNCPoint2[3209] = {X 433.0314, Y 30.5773, Z -2.1667, A 0.000, B 0.000, C 0.000 }
gfCNCPoint2[3210] = {X 432.0739, Y 29.5321, Z -2.1667, A 0.000, B 0.000, C 0.000 }
gfCNCPoint2[3211] = {X 431.2577, Y 28.3733, Z -2.1667, A 0.000, B 0.000, C 0.000 }
gfCNCPoint2[3212] = {X 430.5961, Y 27.1198, Z -2.1667, A 0.000, B 0.000, C 0.000 }
gfCNCPoint2[3213] = {X 430.1000, Y 25.7920, Z -2.1667, A 0.000, B 0.000, C 0.000 }
gfCNCPoint2[3214] = {X 429.6873, Y 24.0071, Z -2.1667, A 0.000, B 0.000, C 0.000 }
gfCNCPoint2[3215] = {X 429.4770, Y 22.1872, Z -2.1667, A 0.000, B 0.000, C 0.000 }
gfCNCPoint2[3216] = {X 429.4719, Y 20.3552, Z -2.1667, A 0.000, B 0.000, C 0.000 }
gfCNCPoint2[3217] = {X 429.6719, Y 18.5342, Z -2.1667, A 0.000, B 0.000, C 0.000 }
gfCNCPoint2[3218] = {X 430.0746, Y 16.7469, Z -2.1667, A 0.000, B 0.000, C 0.000 }
gfCNCPoint2[3219] = {X 430.5853, Y 15.3070, Z -2.1667, A 0.000, B 0.000, C 0.000 }
gfCNCPoint2[3220] = {X 431.2817, Y 13.9471, Z -2.1667, A 0.000, B 0.000, C 0.000 }
gfCNCPoint2[3221] = {X 432.1513, Y 12.6910, Z -2.1667, A 0.000, B 0.000, C 0.000 }
gfCNCPoint2[3222] = {X 433.1792, Y 11.5606, Z -2.1667, A 0.000, B 0.000, C 0.000 }
gfCNCPoint2[3223] = {X 434.3472, Y 10.5757, Z -2.1667, A 0.000, B 0.000, C 0.000 }
gfCNCPoint2[3224] = {X 435.6350, Y 9.7536, Z -2.1667, A 0.000, B 0.000, C 0.000 }
gfCNCPoint2[3225] = {X 437.0200, Y 9.1086, Z -2.1667, A 0.000, B 0.000, C 0.000 }
gfCNCPoint2[3226] = {X 438.4780, Y 8.6520, Z -2.1667, A 0.000, B 0.000, C 0.000 }
gfCNCPoint2[3227] = {X 440.0845, Y 8.3467, Z -2.1667, A 0.000, B 0.000, C 0.000 }
gfCNCPoint2[3228] = {X 441.7098, Y 8.1676, Z -2.1667, A 0.000, B 0.000, C 0.000 }
gfCNCPoint2[3229] = {X 443.3442, Y 8.1156, Z -2.1667, A 0.000, B 0.000, C 0.000 }
gfCNCPoint2[3230] = {X 444.0364, Y 8.1116, Z -2.1667, A 0.000, B 0.000, C 0.000 }
gfCNCPoint2[3231] = {X 459.4465, Y 8.1116, Z -2.1667, A 0.000, B 0.000, C 0.000 }
gfCNCPoint2[3232] = {X 460.3525, Y 8.2136, Z -2.1667, A 0.000, B 0.000, C 0.000 }
gfCNCPoint2[3233] = {X 461.2131, Y 8.5148, Z -2.1667, A 0.000, B 0.000, C 0.000 }
gfCNCPoint2[3234] = {X 461.9850, Y 8.9998, Z -2.1667, A 0.000, B 0.000, C 0.000 }
gfCNCPoint2[3235] = {X 462.6297, Y 9.6445, Z -2.1667, A 0.000, B 0.000, C 0.000 }
gfCNCPoint2[3236] = {X 463.1147, Y 10.4165, Z -2.1667, A 0.000, B 0.000, C 0.000 }
gfCNCPoint2[3237] = {X 463.4159, Y 11.2770, Z -2.1667, A 0.000, B 0.000, C 0.000 }
gfCNCPoint2[3238] = {X 463.5179, Y 12.1830, Z -2.1667, A 0.000, B 0.000, C 0.000 }
gfCNCPoint2[3239] = {X 463.5179, Y 12.9781, Z -2.1667, A 0.000, B 0.000, C 0.000 }
gfCNCPoint2[3240] = {X 463.4240, Y 13.8483, Z -2.1667, A 0.000, B 0.000, C 0.000 }
gfCNCPoint2[3241] = {X 463.1467, Y 14.6784, Z -2.1667, A 0.000, B 0.000, C 0.000 }
gfCNCPoint2[3242] = {X 462.6988, Y 15.4303, Z -2.1667, A 0.000, B 0.000, C 0.000 }
gfCNCPoint2[3243] = {X 462.1007, Y 16.0693, Z -2.1667, A 0.000, B 0.000, C 0.000 }
gfCNCPoint2[3244] = {X 462.0434, Y 16.1178, Z -2.1667, A 0.000, B 0.000, C 0.000 }
gfCNCPoint2[3245] = {X 461.9852, Y 16.1652, Z -2.1667, A 0.000, B 0.000, C 0.000 }
gfCNCPoint2[3246] = {X 461.9897, Y 16.1997, Z -2.1667, A 0.000, B 0.000, C 0.000 }
gfCNCPoint2[3247] = {X 461.9899, Y 28.5936, Z -2.1667, A 0.000, B 0.000, C 0.000 }
gfCNCPoint2[3248] = {X 465.9899, Y 28.5935, Z -2.1667, A 0.000, B 0.000, C 0.000 }
gfCNCPoint2[3249] = {X 465.9899, Y 28.5934, Z -2.1667, A 0.000, B 0.000, C 0.000 }
gfCNCPoint2[3250] = {X 461.9095, Y 28.5936, Z -2.1667, A 0.000, B 0.000, C 0.000 }
gfCNCPoint2[3251] = {X 461.9101, Y 41.0658, Z -2.1667, A 0.000, B 0.000, C 0.000 }
gfCNCPoint2[3252] = {X 462.0490, Y 41.1786, Z -2.1667, A 0.000, B 0.000, C 0.000 }
gfCNCPoint2[3253] = {X 462.6352, Y 41.8051, Z -2.1667, A 0.000, B 0.000, C 0.000 }
gfCNCPoint2[3254] = {X 463.0742, Y 42.5422, Z -2.1667, A 0.000, B 0.000, C 0.000 }
gfCNCPoint2[3255] = {X 463.3460, Y 43.3559, Z -2.1667, A 0.000, B 0.000, C 0.000 }
gfCNCPoint2[3256] = {X 463.4379, Y 44.2089, Z -2.1667, A 0.000, B 0.000, C 0.000 }
gfCNCPoint2[3257] = {X 463.4379, Y 45.0000, Z -2.1667, A 0.000, B 0.000, C 0.000 }
gfCNCPoint2[3258] = {X 463.3377, Y 45.8901, Z -2.1667, A 0.000, B 0.000, C 0.000 }
gfCNCPoint2[3259] = {X 463.0418, Y 46.7355, Z -2.1667, A 0.000, B 0.000, C 0.000 }
gfCNCPoint2[3260] = {X 462.5653, Y 47.4940, Z -2.1667, A 0.000, B 0.000, C 0.000 }
gfCNCPoint2[3261] = {X 461.9319, Y 48.1273, Z -2.1667, A 0.000, B 0.000, C 0.000 }
gfCNCPoint2[3262] = {X 461.1735, Y 48.6039, Z -2.1667, A 0.000, B 0.000, C 0.000 }
gfCNCPoint2[3263] = {X 460.3280, Y 48.8997, Z -2.1667, A 0.000, B 0.000, C 0.000 }
gfCNCPoint2[3264] = {X 459.4379, Y 49.0000, Z -2.1667, A 0.000, B 0.000, C 0.000 }
gfCNCPoint2[3265] = {X 452.9945, Y 49.0000, Z -2.1667, A 0.000, B 0.000, C 0.000 }
gfCNCPoint2[3266] = {X 452.1044, Y 48.8997, Z -2.1667, A 0.000, B 0.000, C 0.000 }
gfCNCPoint2[3267] = {X 451.2589, Y 48.6039, Z -2.1667, A 0.000, B 0.000, C 0.000 }
gfCNCPoint2[3268] = {X 450.5005, Y 48.1273, Z -2.1667, A 0.000, B 0.000, C 0.000 }
gfCNCPoint2[3269] = {X 449.8671, Y 47.4939, Z -2.1667, A 0.000, B 0.000, C 0.000 }
gfCNCPoint2[3270] = {X 449.3906, Y 46.7355, Z -2.1667, A 0.000, B 0.000, C 0.000 }
gfCNCPoint2[3271] = {X 449.0948, Y 45.8900, Z -2.1667, A 0.000, B 0.000, C 0.000 }
gfCNCPoint2[3272] = {X 448.9945, Y 45.0000, Z -2.1667, A 0.000, B 0.000, C 0.000 }
gfCNCPoint2[3273] = {X 448.9949, Y 44.1538, Z -2.1667, A 0.000, B 0.000, C 0.000 }
gfCNCPoint2[3274] = {X 449.1055, Y 43.2730, Z -2.1667, A 0.000, B 0.000, C 0.000 }
gfCNCPoint2[3275] = {X 449.4077, Y 42.4382, Z -2.1667, A 0.000, B 0.000, C 0.000 }
gfCNCPoint2[3276] = {X 449.8865, Y 41.6907, Z -2.1667, A 0.000, B 0.000, C 0.000 }
gfCNCPoint2[3277] = {X 450.5184, Y 41.0672, Z -2.1667, A 0.000, B 0.000, C 0.000 }
gfCNCPoint2[3278] = {X 450.5184, Y 34.1538, Z -2.1667, A 0.000, B 0.000, C 0.000 }
gfCNCPoint2[3279] = {X 447.5225, Y 34.1538, Z -2.1667, A 0.000, B 0.000, C 0.000 }
gfCNCPoint2[3280] = {X 447.2791, Y 34.1524, Z -2.1667, A 0.000, B 0.000, C 0.000 }
gfCNCPoint2[3281] = {X 442.8400, Y 42.7951, Z -2.1667, A 0.000, B 0.000, C 0.000 }
gfCNCPoint2[3282] = {X 442.8965, Y 42.9477, Z -2.1667, A 0.000, B 0.000, C 0.000 }
gfCNCPoint2[3283] = {X 443.0491, Y 43.5701, Z -2.1667, A 0.000, B 0.000, C 0.000 }
gfCNCPoint2[3284] = {X 443.1005, Y 44.2089, Z -2.1667, A 0.000, B 0.000, C 0.000 }
gfCNCPoint2[3285] = {X 443.1005, Y 45.0000, Z -2.1667, A 0.000, B 0.000, C 0.000 }
gfCNCPoint2[3286] = {X 443.0002, Y 45.8901, Z -2.1667, A 0.000, B 0.000, C 0.000 }
gfCNCPoint2[3287] = {X 442.7043, Y 46.7355, Z -2.1667, A 0.000, B 0.000, C 0.000 }
gfCNCPoint2[3288] = {X 442.2278, Y 47.4940, Z -2.1667, A 0.000, B 0.000, C 0.000 }
gfCNCPoint2[3289] = {X 441.5944, Y 48.1273, Z -2.1667, A 0.000, B 0.000, C 0.000 }
gfCNCPoint2[3290] = {X 440.8360, Y 48.6039, Z -2.1667, A 0.000, B 0.000, C 0.000 }
gfCNCPoint2[3291] = {X 439.9906, Y 48.8997, Z -2.1667, A 0.000, B 0.000, C 0.000 }
gfCNCPoint2[3292] = {X 439.1005, Y 49.0000, Z -2.1667, A 0.000, B 0.000, C 0.000 }
gfCNCPoint2[3293] = {X 432.5144, Y 49.0000, Z -2.1667, A 0.000, B 0.000, C 0.000 }
gfCNCPoint2[3294] = {X 431.6243, Y 48.8997, Z -2.1667, A 0.000, B 0.000, C 0.000 }
gfCNCPoint2[3295] = {X 430.7789, Y 48.6039, Z -2.1667, A 0.000, B 0.000, C 0.000 }
gfCNCPoint2[3296] = {X 430.0204, Y 48.1273, Z -2.1667, A 0.000, B 0.000, C 0.000 }
gfCNCPoint2[3297] = {X 429.3871, Y 47.4940, Z -2.1667, A 0.000, B 0.000, C 0.000 }
gfCNCPoint2[3298] = {X 428.9105, Y 46.7355, Z -2.1667, A 0.000, B 0.000, C 0.000 }
gfCNCPoint2[3299] = {X 428.6147, Y 45.8901, Z -2.1667, A 0.000, B 0.000, C 0.000 }
gfCNCPoint2[3300] = {X 428.5144, Y 45.0000, Z -2.1667, A 0.000, B 0.000, C 0.000 }
gfCNCPoint2[3301] = {X 428.5148, Y 44.1538, Z -2.1667, A 0.000, B 0.000, C 0.000 }
gfCNCPoint2[3302] = {X 428.6096, Y 43.3414, Z -2.1667, A 0.000, B 0.000, C 0.000 }
gfCNCPoint2[3303] = {X 428.8676, Y 42.5654, Z -2.1667, A 0.000, B 0.000, C 0.000 }
gfCNCPoint2[3304] = {X 429.2781, Y 41.8580, Z -2.1667, A 0.000, B 0.000, C 0.000 }
gfCNCPoint2[3305] = {X 429.8239, Y 41.2489, Z -2.1667, A 0.000, B 0.000, C 0.000 }
gfCNCPoint2[3306] = {X 430.4821, Y 40.7635, Z -2.1667, A 0.000, B 0.000, C 0.000 }
gfCNCPoint2[3307] = {X 431.2253, Y 40.4222, Z -2.1667, A 0.000, B 0.000, C 0.000 }
gfCNCPoint2[3308] = {X 435.4117, Y 32.2278, Z -2.1667, A 0.000, B 0.000, C 0.000 }
gfCNCPoint2[3309] = {X 434.2137, Y 31.4654, Z -2.1667, A 0.000, B 0.000, C 0.000 }
gfCNCPoint2[3310] = {X 433.1239, Y 30.5551, Z -2.1667, A 0.000, B 0.000, C 0.000 }
gfCNCPoint2[3311] = {X 432.1605, Y 29.5119, Z -2.1667, A 0.000, B 0.000, C 0.000 }
gfCNCPoint2[3312] = {X 431.3394, Y 28.3534, Z -2.1667, A 0.000, B 0.000, C 0.000 }
gfCNCPoint2[3313] = {X 430.6744, Y 27.0987, Z -2.1667, A 0.000, B 0.000, C 0.000 }
gfCNCPoint2[3314] = {X 430.1766, Y 25.7689, Z -2.1667, A 0.000, B 0.000, C 0.000 }
gfCNCPoint2[3315] = {X 429.7660, Y 23.9928, Z -2.1667, A 0.000, B 0.000, C 0.000 }
gfCNCPoint2[3316] = {X 429.5569, Y 22.1819, Z -2.1667, A 0.000, B 0.000, C 0.000 }
gfCNCPoint2[3317] = {X 429.5518, Y 20.3591, Z -2.1667, A 0.000, B 0.000, C 0.000 }
gfCNCPoint2[3318] = {X 429.7509, Y 18.5471, Z -2.1667, A 0.000, B 0.000, C 0.000 }
gfCNCPoint2[3319] = {X 430.1515, Y 16.7687, Z -2.1667, A 0.000, B 0.000, C 0.000 }
gfCNCPoint2[3320] = {X 430.6588, Y 15.3388, Z -2.1667, A 0.000, B 0.000, C 0.000 }
gfCNCPoint2[3321] = {X 431.3503, Y 13.9883, Z -2.1667, A 0.000, B 0.000, C 0.000 }
gfCNCPoint2[3322] = {X 432.2139, Y 12.7408, Z -2.1667, A 0.000, B 0.000, C 0.000 }
gfCNCPoint2[3323] = {X 433.2347, Y 11.6182, Z -2.1667, A 0.000, B 0.000, C 0.000 }
gfCNCPoint2[3324] = {X 434.3946, Y 10.6402, Z -2.1667, A 0.000, B 0.000, C 0.000 }
gfCNCPoint2[3325] = {X 435.6735, Y 9.8237, Z -2.1667, A 0.000, B 0.000, C 0.000 }
gfCNCPoint2[3326] = {X 437.0489, Y 9.1832, Z -2.1667, A 0.000, B 0.000, C 0.000 }
gfCNCPoint2[3327] = {X 438.4968, Y 8.7297, Z -2.1667, A 0.000, B 0.000, C 0.000 }
gfCNCPoint2[3328] = {X 440.0970, Y 8.4257, Z -2.1667, A 0.000, B 0.000, C 0.000 }
gfCNCPoint2[3329] = {X 441.7161, Y 8.2473, Z -2.1667, A 0.000, B 0.000, C 0.000 }
gfCNCPoint2[3330] = {X 443.3442, Y 8.1956, Z -2.1667, A 0.000, B 0.000, C 0.000 }
gfCNCPoint2[3331] = {X 444.0367, Y 8.1916, Z -2.1667, A 0.000, B 0.000, C 0.000 }
gfCNCPoint2[3332] = {X 459.4465, Y 8.1916, Z -2.1667, A 0.000, B 0.000, C 0.000 }
gfCNCPoint2[3333] = {X 460.3347, Y 8.2916, Z -2.1667, A 0.000, B 0.000, C 0.000 }
gfCNCPoint2[3334] = {X 461.1783, Y 8.5868, Z -2.1667, A 0.000, B 0.000, C 0.000 }
gfCNCPoint2[3335] = {X 461.9351, Y 9.0624, Z -2.1667, A 0.000, B 0.000, C 0.000 }
gfCNCPoint2[3336] = {X 462.5671, Y 9.6944, Z -2.1667, A 0.000, B 0.000, C 0.000 }
gfCNCPoint2[3337] = {X 463.0427, Y 10.4512, Z -2.1667, A 0.000, B 0.000, C 0.000 }
gfCNCPoint2[3338] = {X 463.3379, Y 11.2948, Z -2.1667, A 0.000, B 0.000, C 0.000 }
gfCNCPoint2[3339] = {X 463.4379, Y 12.1830, Z -2.1667, A 0.000, B 0.000, C 0.000 }
gfCNCPoint2[3340] = {X 463.4378, Y 13.0163, Z -2.1667, A 0.000, B 0.000, C 0.000 }
gfCNCPoint2[3341] = {X 463.3397, Y 13.8592, Z -2.1667, A 0.000, B 0.000, C 0.000 }
gfCNCPoint2[3342] = {X 463.0660, Y 14.6624, Z -2.1667, A 0.000, B 0.000, C 0.000 }
gfCNCPoint2[3343] = {X 462.6291, Y 15.3898, Z -2.1667, A 0.000, B 0.000, C 0.000 }
gfCNCPoint2[3344] = {X 462.0485, Y 16.0087, Z -2.1667, A 0.000, B 0.000, C 0.000 }
gfCNCPoint2[3345] = {X 461.9721, Y 16.0728, Z -2.1667, A 0.000, B 0.000, C 0.000 }
gfCNCPoint2[3346] = {X 461.8942, Y 16.1351, Z -2.1667, A 0.000, B 0.000, C 0.000 }
gfCNCPoint2[3347] = {X 461.9097, Y 16.1925, Z -2.1667, A 0.000, B 0.000, C 0.000 }
gfCNCPoint2[3348] = {X 461.9090, Y 16.7687, Z -2.1667, A 0.000, B 0.000, C 0.000 }
gfCNCPoint2[3349] = {X 461.9095, Y 28.5936, Z -2.1667, A 0.000, B 0.000, C 0.000 }
gfCNCPoint2[3350] = {X 465.9899, Y 28.5934, Z -2.1667, A 0.000, B 0.000, C 0.000 }
gfCNCPoint2[3351] = {X 465.9899, Y 28.5934, Z 0.8333, A 0.000, B 0.000, C 0.000 }
gfCNCPoint2[3352] = {X 465.9899, Y 28.5934, Z 11.0000, A 0.000, B 0.000, C 0.000 }
gfCNCPoint2[3353] = {X 492.3824, Y 3.7916, Z 11.0000, A 0.000, B 0.000, C 0.000 }
gfCNCPoint2[3354] = {X 492.3824, Y 3.7916, Z 0.8333, A 0.000, B 0.000, C 0.000 }
gfCNCPoint2[3355] = {X 492.3824, Y 3.7916, Z -2.1667, A 0.000, B 0.000, C 0.000 }
gfCNCPoint2[3356] = {X 492.3824, Y 7.8716, Z -2.1667, A 0.000, B 0.000, C 0.000 }
gfCNCPoint2[3357] = {X 502.2066, Y 7.8716, Z -2.1667, A 0.000, B 0.000, C 0.000 }
gfCNCPoint2[3358] = {X 502.7373, Y 7.8757, Z -2.1667, A 0.000, B 0.000, C 0.000 }
gfCNCPoint2[3359] = {X 503.6897, Y 7.9900, Z -2.1667, A 0.000, B 0.000, C 0.000 }
gfCNCPoint2[3360] = {X 504.5931, Y 8.3124, Z -2.1667, A 0.000, B 0.000, C 0.000 }
gfCNCPoint2[3361] = {X 505.4027, Y 8.8268, Z -2.1667, A 0.000, B 0.000, C 0.000 }
gfCNCPoint2[3362] = {X 506.0783, Y 9.5077, Z -2.1667, A 0.000, B 0.000, C 0.000 }
gfCNCPoint2[3363] = {X 506.5863, Y 10.3212, Z -2.1667, A 0.000, B 0.000, C 0.000 }
gfCNCPoint2[3364] = {X 506.9016, Y 11.2271, Z -2.1667, A 0.000, B 0.000, C 0.000 }
gfCNCPoint2[3365] = {X 507.0085, Y 12.1804, Z -2.1667, A 0.000, B 0.000, C 0.000 }
gfCNCPoint2[3366] = {X 507.0085, Y 12.9781, Z -2.1667, A 0.000, B 0.000, C 0.000 }
gfCNCPoint2[3367] = {X 506.9071, Y 13.9083, Z -2.1667, A 0.000, B 0.000, C 0.000 }
gfCNCPoint2[3368] = {X 506.6078, Y 14.7949, Z -2.1667, A 0.000, B 0.000, C 0.000 }
gfCNCPoint2[3369] = {X 506.1247, Y 15.5962, Z -2.1667, A 0.000, B 0.000, C 0.000 }
gfCNCPoint2[3370] = {X 505.4803, Y 16.2747, Z -2.1667, A 0.000, B 0.000, C 0.000 }
gfCNCPoint2[3371] = {X 505.4802, Y 40.9120, Z -2.1667, A 0.000, B 0.000, C 0.000 }
gfCNCPoint2[3372] = {X 506.1190, Y 41.5831, Z -2.1667, A 0.000, B 0.000, C 0.000 }
gfCNCPoint2[3373] = {X 506.5999, Y 42.3749, Z -2.1667, A 0.000, B 0.000, C 0.000 }
gfCNCPoint2[3374] = {X 506.9010, Y 43.2511, Z -2.1667, A 0.000, B 0.000, C 0.000 }
gfCNCPoint2[3375] = {X 507.0083, Y 44.1713, Z -2.1667, A 0.000, B 0.000, C 0.000 }
gfCNCPoint2[3376] = {X 507.0085, Y 45.0000, Z -2.1667, A 0.000, B 0.000, C 0.000 }
gfCNCPoint2[3377] = {X 506.9002, Y 45.9613, Z -2.1667, A 0.000, B 0.000, C 0.000 }
gfCNCPoint2[3378] = {X 506.5807, Y 46.8744, Z -2.1667, A 0.000, B 0.000, C 0.000 }
gfCNCPoint2[3379] = {X 506.0660, Y 47.6935, Z -2.1667, A 0.000, B 0.000, C 0.000 }
gfCNCPoint2[3380] = {X 505.3820, Y 48.3775, Z -2.1667, A 0.000, B 0.000, C 0.000 }
gfCNCPoint2[3381] = {X 504.5629, Y 48.8922, Z -2.1667, A 0.000, B 0.000, C 0.000 }
gfCNCPoint2[3382] = {X 503.6498, Y 49.2117, Z -2.1667, A 0.000, B 0.000, C 0.000 }
gfCNCPoint2[3383] = {X 502.6885, Y 49.3200, Z -2.1667, A 0.000, B 0.000, C 0.000 }
gfCNCPoint2[3384] = {X 496.2450, Y 49.3200, Z -2.1667, A 0.000, B 0.000, C 0.000 }
gfCNCPoint2[3385] = {X 495.2885, Y 49.2128, Z -2.1667, A 0.000, B 0.000, C 0.000 }
gfCNCPoint2[3386] = {X 494.3794, Y 48.8964, Z -2.1667, A 0.000, B 0.000, C 0.000 }
gfCNCPoint2[3387] = {X 493.5630, Y 48.3866, Z -2.1667, A 0.000, B 0.000, C 0.000 }
gfCNCPoint2[3388] = {X 492.8797, Y 47.7087, Z -2.1667, A 0.000, B 0.000, C 0.000 }
gfCNCPoint2[3389] = {X 492.3635, Y 46.8963, Z -2.1667, A 0.000, B 0.000, C 0.000 }
gfCNCPoint2[3390] = {X 492.0399, Y 45.9898, Z -2.1667, A 0.000, B 0.000, C 0.000 }
gfCNCPoint2[3391] = {X 491.9252, Y 45.0341, Z -2.1667, A 0.000, B 0.000, C 0.000 }
gfCNCPoint2[3392] = {X 491.9254, Y 44.1494, Z -2.1667, A 0.000, B 0.000, C 0.000 }
gfCNCPoint2[3393] = {X 492.0359, Y 43.2364, Z -2.1667, A 0.000, B 0.000, C 0.000 }
gfCNCPoint2[3394] = {X 492.3371, Y 42.3675, Z -2.1667, A 0.000, B 0.000, C 0.000 }
gfCNCPoint2[3395] = {X 492.8153, Y 41.5821, Z -2.1667, A 0.000, B 0.000, C 0.000 }
gfCNCPoint2[3396] = {X 493.4490, Y 40.9157, Z -2.1667, A 0.000, B 0.000, C 0.000 }
gfCNCPoint2[3397] = {X 493.4490, Y 34.4738, Z -2.1667, A 0.000, B 0.000, C 0.000 }
gfCNCPoint2[3398] = {X 490.7235, Y 34.4738, Z -2.1667, A 0.000, B 0.000, C 0.000 }
gfCNCPoint2[3399] = {X 486.4397, Y 42.8157, Z -2.1667, A 0.000, B 0.000, C 0.000 }
gfCNCPoint2[3400] = {X 486.4447, Y 42.8289, Z -2.1667, A 0.000, B 0.000, C 0.000 }
gfCNCPoint2[3401] = {X 486.6109, Y 43.4905, Z -2.1667, A 0.000, B 0.000, C 0.000 }
gfCNCPoint2[3402] = {X 486.6708, Y 44.1699, Z -2.1667, A 0.000, B 0.000, C 0.000 }
gfCNCPoint2[3403] = {X 486.6710, Y 45.0000, Z -2.1667, A 0.000, B 0.000, C 0.000 }
gfCNCPoint2[3404] = {X 486.5627, Y 45.9613, Z -2.1667, A 0.000, B 0.000, C 0.000 }
gfCNCPoint2[3405] = {X 486.2432, Y 46.8744, Z -2.1667, A 0.000, B 0.000, C 0.000 }
gfCNCPoint2[3406] = {X 485.7285, Y 47.6935, Z -2.1667, A 0.000, B 0.000, C 0.000 }
gfCNCPoint2[3407] = {X 485.0445, Y 48.3775, Z -2.1667, A 0.000, B 0.000, C 0.000 }
gfCNCPoint2[3408] = {X 484.2254, Y 48.8922, Z -2.1667, A 0.000, B 0.000, C 0.000 }
gfCNCPoint2[3409] = {X 483.3123, Y 49.2117, Z -2.1667, A 0.000, B 0.000, C 0.000 }
gfCNCPoint2[3410] = {X 482.3510, Y 49.3200, Z -2.1667, A 0.000, B 0.000, C 0.000 }
gfCNCPoint2[3411] = {X 475.7650, Y 49.3200, Z -2.1667, A 0.000, B 0.000, C 0.000 }
gfCNCPoint2[3412] = {X 474.8037, Y 49.2117, Z -2.1667, A 0.000, B 0.000, C 0.000 }
gfCNCPoint2[3413] = {X 473.8906, Y 48.8922, Z -2.1667, A 0.000, B 0.000, C 0.000 }
gfCNCPoint2[3414] = {X 473.0715, Y 48.3775, Z -2.1667, A 0.000, B 0.000, C 0.000 }
gfCNCPoint2[3415] = {X 472.3875, Y 47.6935, Z -2.1667, A 0.000, B 0.000, C 0.000 }
gfCNCPoint2[3416] = {X 471.8728, Y 46.8745, Z -2.1667, A 0.000, B 0.000, C 0.000 }
gfCNCPoint2[3417] = {X 471.5533, Y 45.9614, Z -2.1667, A 0.000, B 0.000, C 0.000 }
gfCNCPoint2[3418] = {X 471.4450, Y 45.0001, Z -2.1667, A 0.000, B 0.000, C 0.000 }
gfCNCPoint2[3419] = {X 471.4454, Y 44.1494, Z -2.1667, A 0.000, B 0.000, C 0.000 }
gfCNCPoint2[3420] = {X 471.5430, Y 43.2935, Z -2.1667, A 0.000, B 0.000, C 0.000 }
gfCNCPoint2[3421] = {X 471.8086, Y 42.4740, Z -2.1667, A 0.000, B 0.000, C 0.000 }
gfCNCPoint2[3422] = {X 472.2314, Y 41.7236, Z -2.1667, A 0.000, B 0.000, C 0.000 }
gfCNCPoint2[3423] = {X 472.7947, Y 41.0719, Z -2.1667, A 0.000, B 0.000, C 0.000 }
gfCNCPoint2[3424] = {X 473.4762, Y 40.5449, Z -2.1667, A 0.000, B 0.000, C 0.000 }
gfCNCPoint2[3425] = {X 474.2486, Y 40.1637, Z -2.1667, A 0.000, B 0.000, C 0.000 }
gfCNCPoint2[3426] = {X 478.2331, Y 32.3645, Z -2.1667, A 0.000, B 0.000, C 0.000 }
gfCNCPoint2[3427] = {X 476.9699, Y 31.4967, Z -2.1667, A 0.000, B 0.000, C 0.000 }
gfCNCPoint2[3428] = {X 475.8336, Y 30.4683, Z -2.1667, A 0.000, B 0.000, C 0.000 }
gfCNCPoint2[3429] = {X 474.8446, Y 29.2976, Z -2.1667, A 0.000, B 0.000, C 0.000 }
gfCNCPoint2[3430] = {X 474.0204, Y 28.0055, Z -2.1667, A 0.000, B 0.000, C 0.000 }
gfCNCPoint2[3431] = {X 473.3759, Y 26.6150, Z -2.1667, A 0.000, B 0.000, C 0.000 }
gfCNCPoint2[3432] = {X 472.9225, Y 25.1511, Z -2.1667, A 0.000, B 0.000, C 0.000 }
gfCNCPoint2[3433] = {X 472.6085, Y 23.4680, Z -2.1667, A 0.000, B 0.000, C 0.000 }
gfCNCPoint2[3434] = {X 472.4681, Y 21.7616, Z -2.1667, A 0.000, B 0.000, C 0.000 }
gfCNCPoint2[3435] = {X 472.5028, Y 20.0498, Z -2.1667, A 0.000, B 0.000, C 0.000 }
gfCNCPoint2[3436] = {X 472.7122, Y 18.3505, Z -2.1667, A 0.000, B 0.000, C 0.000 }
gfCNCPoint2[3437] = {X 473.0942, Y 16.6815, Z -2.1667, A 0.000, B 0.000, C 0.000 }
gfCNCPoint2[3438] = {X 473.6374, Y 15.1671, Z -2.1667, A 0.000, B 0.000, C 0.000 }
gfCNCPoint2[3439] = {X 474.3809, Y 13.7404, Z -2.1667, A 0.000, B 0.000, C 0.000 }
gfCNCPoint2[3440] = {X 475.3110, Y 12.4277, Z -2.1667, A 0.000, B 0.000, C 0.000 }
gfCNCPoint2[3441] = {X 476.4105, Y 11.2532, Z -2.1667, A 0.000, B 0.000, C 0.000 }
gfCNCPoint2[3442] = {X 477.6591, Y 10.2387, Z -2.1667, A 0.000, B 0.000, C 0.000 }
gfCNCPoint2[3443] = {X 479.0338, Y 9.4028, Z -2.1667, A 0.000, B 0.000, C 0.000 }
gfCNCPoint2[3444] = {X 480.5090, Y 8.7610, Z -2.1667, A 0.000, B 0.000, C 0.000 }
gfCNCPoint2[3445] = {X 482.0577, Y 8.3252, Z -2.1667, A 0.000, B 0.000, C 0.000 }
gfCNCPoint2[3446] = {X 484.1551, Y 7.9989, Z -2.1667, A 0.000, B 0.000, C 0.000 }
gfCNCPoint2[3447] = {X 486.2746, Y 7.8837, Z -2.1667, A 0.000, B 0.000, C 0.000 }
gfCNCPoint2[3448] = {X 486.9679, Y 7.8716, Z -2.1667, A 0.000, B 0.000, C 0.000 }
gfCNCPoint2[3449] = {X 492.3824, Y 7.8716, Z -2.1667, A 0.000, B 0.000, C 0.000 }
gfCNCPoint2[3450] = {X 492.3824, Y 3.8716, Z -2.1667, A 0.000, B 0.000, C 0.000 }
gfCNCPoint2[3451] = {X 492.3824, Y 7.9516, Z -2.1667, A 0.000, B 0.000, C 0.000 }
gfCNCPoint2[3452] = {X 502.2063, Y 7.9516, Z -2.1667, A 0.000, B 0.000, C 0.000 }
gfCNCPoint2[3453] = {X 502.7367, Y 7.9557, Z -2.1667, A 0.000, B 0.000, C 0.000 }
gfCNCPoint2[3454] = {X 503.6714, Y 8.0679, Z -2.1667, A 0.000, B 0.000, C 0.000 }
gfCNCPoint2[3455] = {X 504.5580, Y 8.3843, Z -2.1667, A 0.000, B 0.000, C 0.000 }
gfCNCPoint2[3456] = {X 505.3525, Y 8.8891, Z -2.1667, A 0.000, B 0.000, C 0.000 }
gfCNCPoint2[3457] = {X 506.0156, Y 9.5573, Z -2.1667, A 0.000, B 0.000, C 0.000 }
gfCNCPoint2[3458] = {X 506.5142, Y 10.3558, Z -2.1667, A 0.000, B 0.000, C 0.000 }
gfCNCPoint2[3459] = {X 506.8236, Y 11.2449, Z -2.1667, A 0.000, B 0.000, C 0.000 }
gfCNCPoint2[3460] = {X 506.9285, Y 12.1804, Z -2.1667, A 0.000, B 0.000, C 0.000 }
gfCNCPoint2[3461] = {X 506.9285, Y 12.9781, Z -2.1667, A 0.000, B 0.000, C 0.000 }
gfCNCPoint2[3462] = {X 506.8270, Y 13.9001, Z -2.1667, A 0.000, B 0.000, C 0.000 }
gfCNCPoint2[3463] = {X 506.5275, Y 14.7780, Z -2.1667, A 0.000, B 0.000, C 0.000 }
gfCNCPoint2[3464] = {X 506.0442, Y 15.5697, Z -2.1667, A 0.000, B 0.000, C 0.000 }
gfCNCPoint2[3465] = {X 505.4003, Y 16.2374, Z -2.1667, A 0.000, B 0.000, C 0.000 }
gfCNCPoint2[3466] = {X 505.4002, Y 40.9501, Z -2.1667, A 0.000, B 0.000, C 0.000 }
gfCNCPoint2[3467] = {X 505.4285, Y 40.9731, Z -2.1667, A 0.000, B 0.000, C 0.000 }
gfCNCPoint2[3468] = {X 506.0554, Y 41.6317, Z -2.1667, A 0.000, B 0.000, C 0.000 }
gfCNCPoint2[3469] = {X 506.5275, Y 42.4089, Z -2.1667, A 0.000, B 0.000, C 0.000 }
gfCNCPoint2[3470] = {X 506.8230, Y 43.2688, Z -2.1667, A 0.000, B 0.000, C 0.000 }
gfCNCPoint2[3471] = {X 506.9283, Y 44.1720, Z -2.1667, A 0.000, B 0.000, C 0.000 }
gfCNCPoint2[3472] = {X 506.9285, Y 45.0000, Z -2.1667, A 0.000, B 0.000, C 0.000 }
gfCNCPoint2[3473] = {X 506.8222, Y 45.9435, Z -2.1667, A 0.000, B 0.000, C 0.000 }
gfCNCPoint2[3474] = {X 506.5086, Y 46.8397, Z -2.1667, A 0.000, B 0.000, C 0.000 }
gfCNCPoint2[3475] = {X 506.0035, Y 47.6436, Z -2.1667, A 0.000, B 0.000, C 0.000 }
gfCNCPoint2[3476] = {X 505.3321, Y 48.3150, Z -2.1667, A 0.000, B 0.000, C 0.000 }
gfCNCPoint2[3477] = {X 504.5282, Y 48.8201, Z -2.1667, A 0.000, B 0.000, C 0.000 }
gfCNCPoint2[3478] = {X 503.6320, Y 49.1337, Z -2.1667, A 0.000, B 0.000, C 0.000 }
gfCNCPoint2[3479] = {X 502.6885, Y 49.2400, Z -2.1667, A 0.000, B 0.000, C 0.000 }
gfCNCPoint2[3480] = {X 496.2450, Y 49.2400, Z -2.1667, A 0.000, B 0.000, C 0.000 }
gfCNCPoint2[3481] = {X 495.3062, Y 49.1348, Z -2.1667, A 0.000, B 0.000, C 0.000 }
gfCNCPoint2[3482] = {X 494.4140, Y 48.8242, Z -2.1667, A 0.000, B 0.000, C 0.000 }
gfCNCPoint2[3483] = {X 493.6127, Y 48.3239, Z -2.1667, A 0.000, B 0.000, C 0.000 }
gfCNCPoint2[3484] = {X 492.9420, Y 47.6585, Z -2.1667, A 0.000, B 0.000, C 0.000 }
gfCNCPoint2[3485] = {X 492.4354, Y 46.8612, Z -2.1667, A 0.000, B 0.000, C 0.000 }
gfCNCPoint2[3486] = {X 492.1178, Y 45.9714, Z -2.1667, A 0.000, B 0.000, C 0.000 }
gfCNCPoint2[3487] = {X 492.0052, Y 45.0335, Z -2.1667, A 0.000, B 0.000, C 0.000 }
gfCNCPoint2[3488] = {X 492.0054, Y 44.1505, Z -2.1667, A 0.000, B 0.000, C 0.000 }
gfCNCPoint2[3489] = {X 492.1159, Y 43.2454, Z -2.1667, A 0.000, B 0.000, C 0.000 }
gfCNCPoint2[3490] = {X 492.4173, Y 42.3850, Z -2.1667, A 0.000, B 0.000, C 0.000 }
gfCNCPoint2[3491] = {X 492.8957, Y 41.6088, Z -2.1667, A 0.000, B 0.000, C 0.000 }
gfCNCPoint2[3492] = {X 493.5290, Y 40.9529, Z -2.1667, A 0.000, B 0.000, C 0.000 }
gfCNCPoint2[3493] = {X 493.5290, Y 34.3938, Z -2.1667, A 0.000, B 0.000, C 0.000 }
gfCNCPoint2[3494] = {X 490.6746, Y 34.3938, Z -2.1667, A 0.000, B 0.000, C 0.000 }
gfCNCPoint2[3495] = {X 486.3522, Y 42.8109, Z -2.1667, A 0.000, B 0.000, C 0.000 }
gfCNCPoint2[3496] = {X 486.3694, Y 42.8560, Z -2.1667, A 0.000, B 0.000, C 0.000 }
gfCNCPoint2[3497] = {X 486.5321, Y 43.5045, Z -2.1667, A 0.000, B 0.000, C 0.000 }
gfCNCPoint2[3498] = {X 486.5908, Y 44.1706, Z -2.1667, A 0.000, B 0.000, C 0.000 }
gfCNCPoint2[3499] = {X 486.5910, Y 45.0000, Z -2.1667, A 0.000, B 0.000, C 0.000 }
gfCNCPoint2[3500] = {X 486.4847, Y 45.9435, Z -2.1667, A 0.000, B 0.000, C 0.000 }
gfCNCPoint2[3501] = {X 486.1711, Y 46.8397, Z -2.1667, A 0.000, B 0.000, C 0.000 }
gfCNCPoint2[3502] = {X 485.6660, Y 47.6436, Z -2.1667, A 0.000, B 0.000, C 0.000 }
gfCNCPoint2[3503] = {X 484.9946, Y 48.3150, Z -2.1667, A 0.000, B 0.000, C 0.000 }
gfCNCPoint2[3504] = {X 484.1907, Y 48.8201, Z -2.1667, A 0.000, B 0.000, C 0.000 }
gfCNCPoint2[3505] = {X 483.2945, Y 49.1337, Z -2.1667, A 0.000, B 0.000, C 0.000 }
gfCNCPoint2[3506] = {X 482.3510, Y 49.2400, Z -2.1667, A 0.000, B 0.000, C 0.000 }
gfCNCPoint2[3507] = {X 475.7650, Y 49.2400, Z -2.1667, A 0.000, B 0.000, C 0.000 }
gfCNCPoint2[3508] = {X 474.8215, Y 49.1337, Z -2.1667, A 0.000, B 0.000, C 0.000 }
gfCNCPoint2[3509] = {X 473.9253, Y 48.8201, Z -2.1667, A 0.000, B 0.000, C 0.000 }
gfCNCPoint2[3510] = {X 473.1214, Y 48.3150, Z -2.1667, A 0.000, B 0.000, C 0.000 }
gfCNCPoint2[3511] = {X 472.4500, Y 47.6436, Z -2.1667, A 0.000, B 0.000, C 0.000 }
gfCNCPoint2[3512] = {X 471.9449, Y 46.8397, Z -2.1667, A 0.000, B 0.000, C 0.000 }
gfCNCPoint2[3513] = {X 471.6313, Y 45.9436, Z -2.1667, A 0.000, B 0.000, C 0.000 }
gfCNCPoint2[3514] = {X 471.5250, Y 45.0001, Z -2.1667, A 0.000, B 0.000, C 0.000 }
gfCNCPoint2[3515] = {X 471.5254, Y 44.1505, Z -2.1667, A 0.000, B 0.000, C 0.000 }
gfCNCPoint2[3516] = {X 471.6223, Y 43.3054, Z -2.1667, A 0.000, B 0.000, C 0.000 }
gfCNCPoint2[3517] = {X 471.8860, Y 42.4967, Z -2.1667, A 0.000, B 0.000, C 0.000 }
gfCNCPoint2[3518] = {X 472.3057, Y 41.7570, Z -2.1667, A 0.000, B 0.000, C 0.000 }
gfCNCPoint2[3519] = {X 472.8647, Y 41.1158, Z -2.1667, A 0.000, B 0.000, C 0.000 }
gfCNCPoint2[3520] = {X 473.5404, Y 40.5992, Z -2.1667, A 0.000, B 0.000, C 0.000 }
gfCNCPoint2[3521] = {X 474.3057, Y 40.2278, Z -2.1667, A 0.000, B 0.000, C 0.000 }
gfCNCPoint2[3522] = {X 478.3386, Y 32.3338, Z -2.1667, A 0.000, B 0.000, C 0.000 }
gfCNCPoint2[3523] = {X 477.0687, Y 31.4726, Z -2.1667, A 0.000, B 0.000, C 0.000 }
gfCNCPoint2[3524] = {X 475.9260, Y 30.4486, Z -2.1667, A 0.000, B 0.000, C 0.000 }
gfCNCPoint2[3525] = {X 474.9313, Y 29.2803, Z -2.1667, A 0.000, B 0.000, C 0.000 }
gfCNCPoint2[3526] = {X 474.1026, Y 27.9889, Z -2.1667, A 0.000, B 0.000, C 0.000 }
gfCNCPoint2[3527] = {X 473.4550, Y 26.5979, Z -2.1667, A 0.000, B 0.000, C 0.000 }
gfCNCPoint2[3528] = {X 473.0002, Y 25.1324, Z -2.1667, A 0.000, B 0.000, C 0.000 }
gfCNCPoint2[3529] = {X 472.6878, Y 23.4574, Z -2.1667, A 0.000, B 0.000, C 0.000 }
gfCNCPoint2[3530] = {X 472.5481, Y 21.7591, Z -2.1667, A 0.000, B 0.000, C 0.000 }
gfCNCPoint2[3531] = {X 472.5826, Y 20.0555, Z -2.1667, A 0.000, B 0.000, C 0.000 }
gfCNCPoint2[3532] = {X 472.7910, Y 18.3643, Z -2.1667, A 0.000, B 0.000, C 0.000 }
gfCNCPoint2[3533] = {X 473.1711, Y 16.7033, Z -2.1667, A 0.000, B 0.000, C 0.000 }
gfCNCPoint2[3534] = {X 473.7107, Y 15.1992, Z -2.1667, A 0.000, B 0.000, C 0.000 }
gfCNCPoint2[3535] = {X 474.4491, Y 13.7821, Z -2.1667, A 0.000, B 0.000, C 0.000 }
gfCNCPoint2[3536] = {X 475.3730, Y 12.4783, Z -2.1667, A 0.000, B 0.000, C 0.000 }
gfCNCPoint2[3537] = {X 476.4650, Y 11.3117, Z -2.1667, A 0.000, B 0.000, C 0.000 }
gfCNCPoint2[3538] = {X 477.7052, Y 10.3040, Z -2.1667, A 0.000, B 0.000, C 0.000 }
gfCNCPoint2[3539] = {X 479.0706, Y 9.4738, Z -2.1667, A 0.000, B 0.000, C 0.000 }
gfCNCPoint2[3540] = {X 480.5359, Y 8.8364, Z -2.1667, A 0.000, B 0.000, C 0.000 }
gfCNCPoint2[3541] = {X 482.0741, Y 8.4036, Z -2.1667, A 0.000, B 0.000, C 0.000 }
gfCNCPoint2[3542] = {X 484.1638, Y 8.0784, Z -2.1667, A 0.000, B 0.000, C 0.000 }
gfCNCPoint2[3543] = {X 486.2755, Y 7.9637, Z -2.1667, A 0.000, B 0.000, C 0.000 }
gfCNCPoint2[3544] = {X 486.9686, Y 7.9516, Z -2.1667, A 0.000, B 0.000, C 0.000 }
gfCNCPoint2[3545] = {X 492.3824, Y 7.9516, Z -2.1667, A 0.000, B 0.000, C 0.000 }
gfCNCPoint2[3546] = {X 492.3824, Y 3.9516, Z -2.1667, A 0.000, B 0.000, C 0.000 }
gfCNCPoint2[3547] = {X 492.3824, Y 8.0316, Z -2.1667, A 0.000, B 0.000, C 0.000 }
gfCNCPoint2[3548] = {X 502.2059, Y 8.0316, Z -2.1667, A 0.000, B 0.000, C 0.000 }
gfCNCPoint2[3549] = {X 502.7361, Y 8.0357, Z -2.1667, A 0.000, B 0.000, C 0.000 }
gfCNCPoint2[3550] = {X 503.6530, Y 8.1458, Z -2.1667, A 0.000, B 0.000, C 0.000 }
gfCNCPoint2[3551] = {X 504.5229, Y 8.4561, Z -2.1667, A 0.000, B 0.000, C 0.000 }
gfCNCPoint2[3552] = {X 505.3024, Y 8.9514, Z -2.1667, A 0.000, B 0.000, C 0.000 }
gfCNCPoint2[3553] = {X 505.9529, Y 9.6070, Z -2.1667, A 0.000, B 0.000, C 0.000 }
gfCNCPoint2[3554] = {X 506.4420, Y 10.3903, Z -2.1667, A 0.000, B 0.000, C 0.000 }
gfCNCPoint2[3555] = {X 506.7456, Y 11.2626, Z -2.1667, A 0.000, B 0.000, C 0.000 }
gfCNCPoint2[3556] = {X 506.8485, Y 12.1804, Z -2.1667, A 0.000, B 0.000, C 0.000 }
gfCNCPoint2[3557] = {X 506.8485, Y 12.9781, Z -2.1667, A 0.000, B 0.000, C 0.000 }
gfCNCPoint2[3558] = {X 506.7469, Y 13.8919, Z -2.1667, A 0.000, B 0.000, C 0.000 }
gfCNCPoint2[3559] = {X 506.4470, Y 14.7610, Z -2.1667, A 0.000, B 0.000, C 0.000 }
gfCNCPoint2[3560] = {X 505.9636, Y 15.5430, Z -2.1667, A 0.000, B 0.000, C 0.000 }
gfCNCPoint2[3561] = {X 505.3203, Y 16.1997, Z -2.1667, A 0.000, B 0.000, C 0.000 }
gfCNCPoint2[3562] = {X 505.3202, Y 40.9887, Z -2.1667, A 0.000, B 0.000, C 0.000 }
gfCNCPoint2[3563] = {X 505.3675, Y 41.0262, Z -2.1667, A 0.000, B 0.000, C 0.000 }
gfCNCPoint2[3564] = {X 505.9863, Y 41.6731, Z -2.1667, A 0.000, B 0.000, C 0.000 }
gfCNCPoint2[3565] = {X 506.4525, Y 42.4373, Z -2.1667, A 0.000, B 0.000, C 0.000 }
gfCNCPoint2[3566] = {X 506.7443, Y 43.2836, Z -2.1667, A 0.000, B 0.000, C 0.000 }
gfCNCPoint2[3567] = {X 506.8483, Y 44.1727, Z -2.1667, A 0.000, B 0.000, C 0.000 }
gfCNCPoint2[3568] = {X 506.8485, Y 45.0000, Z -2.1667, A 0.000, B 0.000, C 0.000 }
gfCNCPoint2[3569] = {X 506.7442, Y 45.9257, Z -2.1667, A 0.000, B 0.000, C 0.000 }
gfCNCPoint2[3570] = {X 506.4365, Y 46.8050, Z -2.1667, A 0.000, B 0.000, C 0.000 }
gfCNCPoint2[3571] = {X 505.9409, Y 47.5937, Z -2.1667, A 0.000, B 0.000, C 0.000 }
gfCNCPoint2[3572] = {X 505.2822, Y 48.2524, Z -2.1667, A 0.000, B 0.000, C 0.000 }
gfCNCPoint2[3573] = {X 504.4934, Y 48.7480, Z -2.1667, A 0.000, B 0.000, C 0.000 }
gfCNCPoint2[3574] = {X 503.6142, Y 49.0557, Z -2.1667, A 0.000, B 0.000, C 0.000 }
gfCNCPoint2[3575] = {X 502.6885, Y 49.1600, Z -2.1667, A 0.000, B 0.000, C 0.000 }
gfCNCPoint2[3576] = {X 496.2450, Y 49.1600, Z -2.1667, A 0.000, B 0.000, C 0.000 }
gfCNCPoint2[3577] = {X 495.3239, Y 49.0567, Z -2.1667, A 0.000, B 0.000, C 0.000 }
gfCNCPoint2[3578] = {X 494.4485, Y 48.7521, Z -2.1667, A 0.000, B 0.000, C 0.000 }
gfCNCPoint2[3579] = {X 493.6623, Y 48.2612, Z -2.1667, A 0.000, B 0.000, C 0.000 }
gfCNCPoint2[3580] = {X 493.0043, Y 47.6084, Z -2.1667, A 0.000, B 0.000, C 0.000 }
gfCNCPoint2[3581] = {X 492.5072, Y 46.8261, Z -2.1667, A 0.000, B 0.000, C 0.000 }
gfCNCPoint2[3582] = {X 492.1957, Y 45.9531, Z -2.1667, A 0.000, B 0.000, C 0.000 }
gfCNCPoint2[3583] = {X 492.0852, Y 45.0328, Z -2.1667, A 0.000, B 0.000, C 0.000 }
gfCNCPoint2[3584] = {X 492.0854, Y 44.1516, Z -2.1667, A 0.000, B 0.000, C 0.000 }
gfCNCPoint2[3585] = {X 492.1960, Y 43.2545, Z -2.1667, A 0.000, B 0.000, C 0.000 }
gfCNCPoint2[3586] = {X 492.4976, Y 42.4026, Z -2.1667, A 0.000, B 0.000, C 0.000 }
gfCNCPoint2[3587] = {X 492.9762, Y 41.6358, Z -2.1667, A 0.000, B 0.000, C 0.000 }
gfCNCPoint2[3588] = {X 493.6090, Y 40.9906, Z -2.1667, A 0.000, B 0.000, C 0.000 }
gfCNCPoint2[3589] = {X 493.6090, Y 34.3138, Z -2.1667, A 0.000, B 0.000, C 0.000 }
gfCNCPoint2[3590] = {X 490.6258, Y 34.3138, Z -2.1667, A 0.000, B 0.000, C 0.000 }
gfCNCPoint2[3591] = {X 486.2647, Y 42.8061, Z -2.1667, A 0.000, B 0.000, C 0.000 }
gfCNCPoint2[3592] = {X 486.2941, Y 42.8830, Z -2.1667, A 0.000, B 0.000, C 0.000 }
gfCNCPoint2[3593] = {X 486.4534, Y 43.5186, Z -2.1667, A 0.000, B 0.000, C 0.000 }
gfCNCPoint2[3594] = {X 486.5108, Y 44.1713, Z -2.1667, A 0.000, B 0.000, C 0.000 }
gfCNCPoint2[3595] = {X 486.5110, Y 45.0000, Z -2.1667, A 0.000, B 0.000, C 0.000 }
gfCNCPoint2[3596] = {X 486.4067, Y 45.9257, Z -2.1667, A 0.000, B 0.000, C 0.000 }
gfCNCPoint2[3597] = {X 486.0990, Y 46.8050, Z -2.1667, A 0.000, B 0.000, C 0.000 }
gfCNCPoint2[3598] = {X 485.6034, Y 47.5937, Z -2.1667, A 0.000, B 0.000, C 0.000 }
gfCNCPoint2[3599] = {X 484.9447, Y 48.2524, Z -2.1667, A 0.000, B 0.000, C 0.000 }
gfCNCPoint2[3600] = {X 484.1560, Y 48.7480, Z -2.1667, A 0.000, B 0.000, C 0.000 }
gfCNCPoint2[3601] = {X 483.2767, Y 49.0557, Z -2.1667, A 0.000, B 0.000, C 0.000 }
gfCNCPoint2[3602] = {X 482.3510, Y 49.1600, Z -2.1667, A 0.000, B 0.000, C 0.000 }
gfCNCPoint2[3603] = {X 475.7650, Y 49.1600, Z -2.1667, A 0.000, B 0.000, C 0.000 }
gfCNCPoint2[3604] = {X 474.8393, Y 49.0557, Z -2.1667, A 0.000, B 0.000, C 0.000 }
gfCNCPoint2[3605] = {X 473.9600, Y 48.7480, Z -2.1667, A 0.000, B 0.000, C 0.000 }
gfCNCPoint2[3606] = {X 473.1713, Y 48.2524, Z -2.1667, A 0.000, B 0.000, C 0.000 }
gfCNCPoint2[3607] = {X 472.5126, Y 47.5937, Z -2.1667, A 0.000, B 0.000, C 0.000 }
gfCNCPoint2[3608] = {X 472.0169, Y 46.8050, Z -2.1667, A 0.000, B 0.000, C 0.000 }
gfCNCPoint2[3609] = {X 471.7093, Y 45.9257, Z -2.1667, A 0.000, B 0.000, C 0.000 }
gfCNCPoint2[3610] = {X 471.6050, Y 45.0000, Z -2.1667, A 0.000, B 0.000, C 0.000 }
gfCNCPoint2[3611] = {X 471.6054, Y 44.1516, Z -2.1667, A 0.000, B 0.000, C 0.000 }
gfCNCPoint2[3612] = {X 471.7016, Y 43.3174, Z -2.1667, A 0.000, B 0.000, C 0.000 }
gfCNCPoint2[3613] = {X 471.9634, Y 42.5195, Z -2.1667, A 0.000, B 0.000, C 0.000 }
gfCNCPoint2[3614] = {X 472.3801, Y 41.7905, Z -2.1667, A 0.000, B 0.000, C 0.000 }
gfCNCPoint2[3615] = {X 472.9347, Y 41.1600, Z -2.1667, A 0.000, B 0.000, C 0.000 }
gfCNCPoint2[3616] = {X 473.6046, Y 40.6537, Z -2.1667, A 0.000, B 0.000, C 0.000 }
gfCNCPoint2[3617] = {X 474.3626, Y 40.2923, Z -2.1667, A 0.000, B 0.000, C 0.000 }
gfCNCPoint2[3618] = {X 478.4444, Y 32.3026, Z -2.1667, A 0.000, B 0.000, C 0.000 }
gfCNCPoint2[3619] = {X 477.1677, Y 31.4482, Z -2.1667, A 0.000, B 0.000, C 0.000 }
gfCNCPoint2[3620] = {X 476.0185, Y 30.4287, Z -2.1667, A 0.000, B 0.000, C 0.000 }
gfCNCPoint2[3621] = {X 475.0181, Y 29.2629, Z -2.1667, A 0.000, B 0.000, C 0.000 }
gfCNCPoint2[3622] = {X 474.1848, Y 27.9723, Z -2.1667, A 0.000, B 0.000, C 0.000 }
gfCNCPoint2[3623] = {X 473.5342, Y 26.5807, Z -2.1667, A 0.000, B 0.000, C 0.000 }
gfCNCPoint2[3624] = {X 473.0780, Y 25.1138, Z -2.1667, A 0.000, B 0.000, C 0.000 }
gfCNCPoint2[3625] = {X 472.7671, Y 23.4468, Z -2.1667, A 0.000, B 0.000, C 0.000 }
gfCNCPoint2[3626] = {X 472.6281, Y 21.7567, Z -2.1667, A 0.000, B 0.000, C 0.000 }
gfCNCPoint2[3627] = {X 472.6624, Y 20.0612, Z -2.1667, A 0.000, B 0.000, C 0.000 }
